LIN {X 0,Y 432.389,Z 395.501,A -85,B 0,C 180,E1 -9380.764,E2 -9380.764} C_VEL
LIN {X 0,Y 432.358,Z 395.258,A -85,B 0,C 180,E1 -9380.859,E2 -9380.859} C_VEL
LIN {X 0,Y 432.387,Z 395.255,A -85,B 0,C 180,E1 -9384.463,E2 -9384.463} C_VEL
LIN {X 0,Y 432.394,Z 395.251,A -85,B 0,C 180,E1 -9387.071,E2 -9387.071} C_VEL
LIN {X 0,Y 432.35,Z 395.255,A -85,B 0,C 180,E1 -9390.51,E2 -9390.51} C_VEL
LIN {X 0,Y 432.362,Z 395.254,A -85,B 0,C 180,E1 -9394.003,E2 -9394.003} C_VEL
LIN {X 0,Y 432.325,Z 395.26,A -85,B 0,C 180,E1 -9397.197,E2 -9397.197} C_VEL
LIN {X 0,Y 432.339,Z 395.258,A -85,B 0,C 180,E1 -9400.179,E2 -9400.179} C_VEL
LIN {X 0,Y 432.32,Z 395.262,A -85,B 0,C 180,E1 -9403.06,E2 -9403.06} C_VEL
LIN {X 0,Y 432.405,Z 395.425,A -85,B 0,C 180,E1 -9405.158,E2 -9405.158} C_VEL
LIN {X 0,Y 433.777,Z 402.089,A -85,B 0,C 180,E1 -9408.184,E2 -9408.184} C_VEL
LIN {X 0,Y 434.807,Z 407.668,A -85,B 0,C 180,E1 -9410.323,E2 -9410.323} C_VEL
LIN {X 0,Y 434.807,Z 411.22,A -85,B 0,C 180,E1 -9411.515,E2 -9411.515} C_VEL
LIN {X 0,Y 433.579,Z 424.383,A -85,B 0,C 180,E1 -9415.435,E2 -9415.435} C_VEL
LIN {X 0,Y 433.139,Z 436.415,A -85,B 0,C 180,E1 -9418.719,E2 -9418.719} C_VEL
LIN {X 0,Y 432.871,Z 446.188,A -85,B 0,C 180,E1 -9421.251,E2 -9421.251} C_VEL
LIN {X 0,Y 432.552,Z 460.292,A -85,B 0,C 180,E1 -9424.753,E2 -9424.753} C_VEL
LIN {X 0,Y 432.258,Z 473.917,A -85,B 0,C 180,E1 -9428.04,E2 -9428.04} C_VEL
LIN {X 0,Y 432.199,Z 479.961,A -85,B 0,C 180,E1 -9429.474,E2 -9429.474} C_VEL
LIN {X 0,Y 434.596,Z 497.607,A -85,B 0,C 180,E1 -9430.147,E2 -9430.147} C_VEL
LIN {X 0,Y 435.507,Z 512.403,A -85,B 0,C 180,E1 -9430.82,E2 -9430.82} C_VEL
LIN {X 0,Y 436.409,Z 524.648,A -85,B 0,C 180,E1 -9431.515,E2 -9431.515} C_VEL
LIN {X 0,Y 435.473,Z 538.641,A -85,B 0,C 180,E1 -9432.41,E2 -9432.41} C_VEL
LIN {X 0,Y 434.546,Z 551.621,A -85,B 0,C 180,E1 -9433.437,E2 -9433.437} C_VEL
LIN {X 0,Y 433.58,Z 564.986,A -85,B 0,C 180,E1 -9434.727,E2 -9434.727} C_VEL
LIN {X 0,Y 432.899,Z 577.024,A -85,B 0,C 180,E1 -9436.144,E2 -9436.144} C_VEL
LIN {X 0,Y 432.318,Z 587.05,A -85,B 0,C 180,E1 -9437.569,E2 -9437.569} C_VEL
LIN {X 0,Y 432.076,Z 595.4,A -85,B 0,C 180,E1 -9438.981,E2 -9438.981} C_VEL
LIN {X 0,Y 431.843,Z 603.466,A -85,B 0,C 180,E1 -9440.633,E2 -9440.633} C_VEL
LIN {X 0,Y 431.739,Z 609.158,A -85,B 0,C 180,E1 -9442.046,E2 -9442.046} C_VEL
LIN {X 0,Y 431.725,Z 613.768,A -85,B 0,C 180,E1 -9443.456,E2 -9443.456} C_VEL
LIN {X 0,Y 431.834,Z 618.501,A -85,B 0,C 180,E1 -9445.332,E2 -9445.332} C_VEL
LIN {X 0,Y 431.768,Z 621.63,A -85,B 0,C 180,E1 -9447.2,E2 -9447.2} C_VEL
LIN {X 0,Y 431.795,Z 623.265,A -85,B 0,C 180,E1 -9449.066,E2 -9449.066} C_VEL
LIN {X 0,Y 431.897,Z 623.543,A -85,B 0,C 180,E1 -9449.999,E2 -9449.999} C_VEL
LIN {X 0,Y 431.718,Z 622.951,A -85,B 0,C 180,E1 -9451.865,E2 -9451.865} C_VEL
LIN {X 0,Y 431.718,Z 620.927,A -85,B 0,C 180,E1 -9453.732,E2 -9453.732} C_VEL
LIN {X 0,Y 431.638,Z 617.389,A -85,B 0,C 180,E1 -9455.605,E2 -9455.605} C_VEL
LIN {X 0,Y 431.629,Z 613.716,A -85,B 0,C 180,E1 -9457.013,E2 -9457.013} C_VEL
LIN {X 0,Y 431.673,Z 609.053,A -85,B 0,C 180,E1 -9458.425,E2 -9458.425} C_VEL
LIN {X 0,Y 431.835,Z 602.28,A -85,B 0,C 180,E1 -9460.075,E2 -9460.075} C_VEL
LIN {X 0,Y 432.208,Z 593.835,A -85,B 0,C 180,E1 -9461.726,E2 -9461.726} C_VEL
LIN {X 0,Y 432.652,Z 585.027,A -85,B 0,C 180,E1 -9463.144,E2 -9463.144} C_VEL
LIN {X 0,Y 433.303,Z 574.399,A -85,B 0,C 180,E1 -9464.559,E2 -9464.559} C_VEL
LIN {X 0,Y 434.087,Z 562.586,A -85,B 0,C 180,E1 -9465.854,E2 -9465.854} C_VEL
LIN {X 0,Y 434.998,Z 550.878,A -85,B 0,C 180,E1 -9466.906,E2 -9466.906} C_VEL
LIN {X 0,Y 435.864,Z 538.135,A -85,B 0,C 180,E1 -9467.839,E2 -9467.839} C_VEL
LIN {X 0,Y 436.673,Z 523.959,A -85,B 0,C 180,E1 -9468.654,E2 -9468.654} C_VEL
LIN {X 0,Y 435.13,Z 509.071,A -85,B 0,C 180,E1 -9469.367,E2 -9469.367} C_VEL
LIN {X 0,Y 433.039,Z 493.7,A -85,B 0,C 180,E1 -9469.915,E2 -9469.915} C_VEL
LIN {X 0,Y 432.378,Z 488.684,A -85,B 0,C 180,E1 -9470.081,E2 -9470.081} C_VEL
LIN {X 0,Y 432.86,Z 475.595,A -85,B 0,C 180,E1 -9473.438,E2 -9473.438} C_VEL
LIN {X 0,Y 433.463,Z 461.986,A -85,B 0,C 180,E1 -9476.998,E2 -9476.998} C_VEL
LIN {X 0,Y 434.313,Z 447.187,A -85,B 0,C 180,E1 -9480.947,E2 -9480.947} C_VEL
LIN {X 0,Y 435.145,Z 434.082,A -85,B 0,C 180,E1 -9484.543,E2 -9484.543} C_VEL
LIN {X 0,Y 436.259,Z 419.683,A -85,B 0,C 180,E1 -9488.625,E2 -9488.625} C_VEL
LIN {X 0,Y 436.418,Z 416.038,A -85,B 0,C 180,E1 -9489.689,E2 -9489.689} C_VEL
LIN {X 0,Y 435.184,Z 408.622,A -85,B 0,C 180,E1 -9492.023,E2 -9492.023} C_VEL
LIN {X 0,Y 432.796,Z 397.532,A -85,B 0,C 180,E1 -9495.713,E2 -9495.713} C_VEL
LIN {X 0,Y 432.346,Z 395.255,A -85,B 0,C 180,E1 -9496.543,E2 -9496.543} C_VEL
LIN {X 0,Y 432.352,Z 395.257,A -85,B 0,C 180,E1 -9499.815,E2 -9499.815} C_VEL
LIN {X 0,Y 432.309,Z 395.26,A -85,B 0,C 180,E1 -9503.022,E2 -9503.022} C_VEL
LIN {X 0,Y 432.35,Z 395.253,A -85,B 0,C 180,E1 -9505.996,E2 -9505.996} C_VEL
LIN {X 0,Y 432.385,Z 395.25,A -85,B 0,C 180,E1 -9509.743,E2 -9509.743} C_VEL
LIN {X 0,Y 432.39,Z 395.252,A -85,B 0,C 180,E1 -9513.372,E2 -9513.372} C_VEL
LIN {X 0,Y 432.361,Z 395.251,A -85,B 0,C 180,E1 -9516.023,E2 -9516.023} C_VEL
LIN {X 0,Y 432.34,Z 395.257,A -85,B 0,C 180,E1 -9519.046,E2 -9519.046} C_VEL
LIN {X 0,Y 432.367,Z 395.251,A -85,B 0,C 180,E1 -9522.011,E2 -9522.011} C_VEL
LIN {X 0,Y 432.385,Z 395.251,A -85,B 0,C 180,E1 -9524.926,E2 -9524.926} C_VEL
LIN {X 0,Y 432.47,Z 395.238,A -85,B 0,C 180,E1 -9527.804,E2 -9527.804} C_VEL
LIN {X 0,Y 432.481,Z 395.238,A -85,B 0,C 180,E1 -9531.59,E2 -9531.59} C_VEL
LIN {X 0,Y 432.588,Z 395.225,A -85,B 0,C 180,E1 -9534.406,E2 -9534.406} C_VEL
LIN {X 0,Y 432.596,Z 395.223,A -85,B 0,C 180,E1 -9538.138,E2 -9538.138} C_VEL
LIN {X 0,Y 432.724,Z 395.206,A -85,B 0,C 180,E1 -9540,E2 -9540} C_VEL
LIN {X 0,Y 432.597,Z 395.224,A -85,B 0,C 180,E1 -9542.794,E2 -9542.794} C_VEL
LIN {X 0,Y 432.564,Z 395.228,A -85,B 0,C 180,E1 -9546.531,E2 -9546.531} C_VEL
LIN {X 0,Y 432.435,Z 395.244,A -85,B 0,C 180,E1 -9549.354,E2 -9549.354} C_VEL
LIN {X 0,Y 432.435,Z 395.245,A -85,B 0,C 180,E1 -9552.813,E2 -9552.813} C_VEL
LIN {X 0,Y 432.403,Z 395.248,A -85,B 0,C 180,E1 -9556.48,E2 -9556.48} C_VEL
LIN {X 0,Y 432.33,Z 395.256,A -85,B 0,C 180,E1 -9559.961,E2 -9559.961} C_VEL
LIN {X 0,Y 432.31,Z 395.262,A -85,B 0,C 180,E1 -9562.965,E2 -9562.965} C_VEL
LIN {X 0,Y 432.356,Z 395.253,A -85,B 0,C 180,E1 -9566.033,E2 -9566.033} C_VEL
LIN {X 0,Y 432.335,Z 395.256,A -85,B 0,C 180,E1 -9569.188,E2 -9569.188} C_VEL
LIN {X 0,Y 432.316,Z 395.259,A -85,B 0,C 180,E1 -9572.444,E2 -9572.444} C_VEL
LIN {X 0,Y 432.339,Z 395.254,A -85,B 0,C 180,E1 -9575.633,E2 -9575.633} C_VEL
LIN {X 0,Y 432.346,Z 395.257,A -85,B 0,C 180,E1 -9578.718,E2 -9578.718} C_VEL
LIN {X 0,Y 432.33,Z 395.256,A -85,B 0,C 180,E1 -9581.798,E2 -9581.798} C_VEL
LIN {X 0,Y 432.337,Z 395.256,A -85,B 0,C 180,E1 -9584.347,E2 -9584.347} C_VEL
LIN {X 0,Y 432.316,Z 395.259,A -85,B 0,C 180,E1 -9587.017,E2 -9587.017} C_VEL
LIN {X 0,Y 432.353,Z 395.253,A -85,B 0,C 180,E1 -9589.818,E2 -9589.818} C_VEL
LIN {X 0,Y 432.315,Z 395.259,A -85,B 0,C 180,E1 -9593.025,E2 -9593.025} C_VEL
LIN {X 0,Y 432.357,Z 395.253,A -85,B 0,C 180,E1 -9595.998,E2 -9595.998} C_VEL
LIN {X 0,Y 432.346,Z 395.253,A -85,B 0,C 180,E1 -9599.491,E2 -9599.491} C_VEL
LIN {X 0,Y 432.392,Z 395.249,A -85,B 0,C 180,E1 -9602.93,E2 -9602.93} C_VEL
LIN {X 0,Y 432.372,Z 395.252,A -85,B 0,C 180,E1 -9606.025,E2 -9606.025} C_VEL
LIN {X 0,Y 432.351,Z 395.253,A -85,B 0,C 180,E1 -9609.047,E2 -9609.047} C_VEL
LIN {X 0,Y 432.377,Z 395.251,A -85,B 0,C 180,E1 -9612.012,E2 -9612.012} C_VEL
LIN {X 0,Y 432.314,Z 395.26,A -85,B 0,C 180,E1 -9614.925,E2 -9614.925} C_VEL
LIN {X 0,Y 432.25,Z 395.365,A -85,B 0,C 180,E1 -9616.547,E2 -9616.547} C_VEL
LIN {X 0,Y 436.298,Z 408.442,A -85,B 0,C 180,E1 -9617.107,E2 -9617.107} C_VEL
LIN {X 0,Y 436.567,Z 411.618,A -85,B 0,C 180,E1 -9617.251,E2 -9617.251} C_VEL
LIN {X 0,Y 436.282,Z 423.378,A -85,B 0,C 180,E1 -9617.832,E2 -9617.832} C_VEL
LIN {X 0,Y 435.847,Z 435.168,A -85,B 0,C 180,E1 -9618.609,E2 -9618.609} C_VEL
LIN {X 0,Y 435.323,Z 446.119,A -85,B 0,C 180,E1 -9619.537,E2 -9619.537} C_VEL
LIN {X 0,Y 434.762,Z 455.934,A -85,B 0,C 180,E1 -9620.569,E2 -9620.569} C_VEL
LIN {X 0,Y 434.12,Z 465.767,A -85,B 0,C 180,E1 -9621.858,E2 -9621.858} C_VEL
LIN {X 0,Y 433.656,Z 474.255,A -85,B 0,C 180,E1 -9623.253,E2 -9623.253} C_VEL
LIN {X 0,Y 433.113,Z 481.113,A -85,B 0,C 180,E1 -9624.647,E2 -9624.647} C_VEL
LIN {X 0,Y 432.913,Z 485.709,A -85,B 0,C 180,E1 -9625.812,E2 -9625.812} C_VEL
LIN {X 0,Y 432.731,Z 487.452,A -85,B 0,C 180,E1 -9626.316,E2 -9626.316} C_VEL
LIN {X 0,Y 431.918,Z 489.8,A -85,B 0,C 180,E1 -9627.029,E2 -9627.029} C_VEL
LIN {X 0,Y 427.594,Z 494.515,A -85,B 0,C 180,E1 -9628.67,E2 -9628.67} C_VEL
LIN {X 0,Y 425.543,Z 496.535,A -85,B 0,C 180,E1 -9629.661,E2 -9629.661} C_VEL
LIN {X 0,Y 425.142,Z 497.269,A -85,B 0,C 180,E1 -9630.181,E2 -9630.181} C_VEL
LIN {X 0,Y 425.026,Z 498.178,A -85,B 0,C 180,E1 -9630.948,E2 -9630.948} C_VEL
LIN {X 0,Y 425.094,Z 498.851,A -85,B 0,C 180,E1 -9631.896,E2 -9631.896} C_VEL
LIN {X 0,Y 425.025,Z 499.13,A -85,B 0,C 180,E1 -9633.793,E2 -9633.793} C_VEL
LIN {X 0,Y 425.111,Z 498.668,A -85,B 0,C 180,E1 -9634.742,E2 -9634.742} C_VEL
LIN {X 0,Y 425.3,Z 497.792,A -85,B 0,C 180,E1 -9635.691,E2 -9635.691} C_VEL
LIN {X 0,Y 425.456,Z 494.927,A -85,B 0,C 180,E1 -9637.595,E2 -9637.595} C_VEL
LIN {X 0,Y 425.736,Z 491.621,A -85,B 0,C 180,E1 -9639.024,E2 -9639.024} C_VEL
LIN {X 0,Y 426.167,Z 487.23,A -85,B 0,C 180,E1 -9640.452,E2 -9640.452} C_VEL
LIN {X 0,Y 426.614,Z 480.562,A -85,B 0,C 180,E1 -9642.126,E2 -9642.126} C_VEL
LIN {X 0,Y 426.971,Z 474.618,A -85,B 0,C 180,E1 -9643.324,E2 -9643.324} C_VEL
LIN {X 0,Y 427.736,Z 465.841,A -85,B 0,C 180,E1 -9644.755,E2 -9644.755} C_VEL
LIN {X 0,Y 428.389,Z 455.68,A -85,B 0,C 180,E1 -9646.073,E2 -9646.073} C_VEL
LIN {X 0,Y 428.99,Z 445.34,A -85,B 0,C 180,E1 -9647.152,E2 -9647.152} C_VEL
LIN {X 0,Y 429.538,Z 435.288,A -85,B 0,C 180,E1 -9647.989,E2 -9647.989} C_VEL
LIN {X 0,Y 430.03,Z 423.551,A -85,B 0,C 180,E1 -9648.754,E2 -9648.754} C_VEL
LIN {X 0,Y 430.232,Z 411.232,A -85,B 0,C 180,E1 -9649.362,E2 -9649.362} C_VEL
LIN {X 0,Y 426.035,Z 398.909,A -85,B 0,C 180,E1 -9649.98,E2 -9649.98} C_VEL
LIN {X 0,Y 425.159,Z 396.153,A -85,B 0,C 180,E1 -9650.101,E2 -9650.101} C_VEL
LIN {X 0,Y 425.287,Z 396.134,A -85,B 0,C 180,E1 -9653.367,E2 -9653.367} C_VEL
LIN {X 0,Y 425.361,Z 396.125,A -85,B 0,C 180,E1 -9656.495,E2 -9656.495} C_VEL
LIN {X 0,Y 425.297,Z 396.133,A -85,B 0,C 180,E1 -9659.72,E2 -9659.72} C_VEL
LIN {X 0,Y 425.287,Z 396.139,A -85,B 0,C 180,E1 -9663.048,E2 -9663.048} C_VEL
LIN {X 0,Y 425.287,Z 396.135,A -85,B 0,C 180,E1 -9665.929,E2 -9665.929} C_VEL
LIN {X 0,Y 425.293,Z 396.129,A -85,B 0,C 180,E1 -9669.042,E2 -9669.042} C_VEL
LIN {X 0,Y 425.295,Z 396.132,A -85,B 0,C 180,E1 -9671.958,E2 -9671.958} C_VEL
LIN {X 0,Y 425.295,Z 396.128,A -85,B 0,C 180,E1 -9675.283,E2 -9675.283} C_VEL
LIN {X 0,Y 425.281,Z 396.131,A -85,B 0,C 180,E1 -9678.622,E2 -9678.622} C_VEL
LIN {X 0,Y 425.314,Z 396.108,A -85,B 0,C 180,E1 -9681.103,E2 -9681.103} C_VEL
LIN {X 0,Y 425.306,Z 396.131,A -85,B 0,C 180,E1 -9684.664,E2 -9684.664} C_VEL
LIN {X 0,Y 425.269,Z 396.125,A -85,B 0,C 180,E1 -9688.073,E2 -9688.073} C_VEL
LIN {X 0,Y 425.335,Z 396.103,A -85,B 0,C 180,E1 -9691.368,E2 -9691.368} C_VEL
LIN {X 0,Y 425.358,Z 396.118,A -85,B 0,C 180,E1 -9693.505,E2 -9693.505} C_VEL
LIN {X 0,Y 425.289,Z 396.132,A -85,B 0,C 180,E1 -9696.633,E2 -9696.633} C_VEL
LIN {X 0,Y 425.299,Z 396.135,A -85,B 0,C 180,E1 -9699.694,E2 -9699.694} C_VEL
LIN {X 0,Y 425.329,Z 396.131,A -85,B 0,C 180,E1 -9701.889,E2 -9701.889} C_VEL
LIN {X 0,Y 430.063,Z 411.616,A -85,B 0,C 180,E1 -9703.015,E2 -9703.015} C_VEL
LIN {X 0,Y 430.272,Z 415.083,A -85,B 0,C 180,E1 -9703.268,E2 -9703.268} C_VEL
LIN {X 0,Y 429.619,Z 427.403,A -85,B 0,C 180,E1 -9704.219,E2 -9704.219} C_VEL
LIN {X 0,Y 428.793,Z 440.383,A -85,B 0,C 180,E1 -9705.449,E2 -9705.449} C_VEL
LIN {X 0,Y 428.002,Z 451.242,A -85,B 0,C 180,E1 -9706.709,E2 -9706.709} C_VEL
LIN {X 0,Y 427.252,Z 461.376,A -85,B 0,C 180,E1 -9708.134,E2 -9708.134} C_VEL
LIN {X 0,Y 426.771,Z 469.803,A -85,B 0,C 180,E1 -9709.563,E2 -9709.563} C_VEL
LIN {X 0,Y 426.188,Z 477.894,A -85,B 0,C 180,E1 -9711.226,E2 -9711.226} C_VEL
LIN {X 0,Y 425.775,Z 484.425,A -85,B 0,C 180,E1 -9712.888,E2 -9712.888} C_VEL
LIN {X 0,Y 425.45,Z 490.251,A -85,B 0,C 180,E1 -9714.787,E2 -9714.787} C_VEL
LIN {X 0,Y 425.156,Z 493.572,A -85,B 0,C 180,E1 -9716.208,E2 -9716.208} C_VEL
LIN {X 0,Y 425.096,Z 496.722,A -85,B 0,C 180,E1 -9718.105,E2 -9718.105} C_VEL
LIN {X 0,Y 425.055,Z 498.526,A -85,B 0,C 180,E1 -9720,E2 -9720} C_VEL
LIN {X 0,Y 425.159,Z 498.985,A -85,B 0,C 180,E1 -9721.894,E2 -9721.894} C_VEL
LIN {X 0,Y 425.197,Z 498.132,A -85,B 0,C 180,E1 -9723.791,E2 -9723.791} C_VEL
LIN {X 0,Y 425.467,Z 495.878,A -85,B 0,C 180,E1 -9725.688,E2 -9725.688} C_VEL
LIN {X 0,Y 425.857,Z 492.193,A -85,B 0,C 180,E1 -9727.586,E2 -9727.586} C_VEL
LIN {X 0,Y 426.379,Z 487.005,A -85,B 0,C 180,E1 -9729.487,E2 -9729.487} C_VEL
LIN {X 0,Y 426.836,Z 481.998,A -85,B 0,C 180,E1 -9730.915,E2 -9730.915} C_VEL
LIN {X 0,Y 427.533,Z 474.75,A -85,B 0,C 180,E1 -9732.58,E2 -9732.58} C_VEL
LIN {X 0,Y 428.349,Z 467.101,A -85,B 0,C 180,E1 -9734.005,E2 -9734.005} C_VEL
LIN {X 0,Y 429.177,Z 457.883,A -85,B 0,C 180,E1 -9735.432,E2 -9735.432} C_VEL
LIN {X 0,Y 430.005,Z 447.738,A -85,B 0,C 180,E1 -9736.742,E2 -9736.742} C_VEL
LIN {X 0,Y 430.927,Z 436.514,A -85,B 0,C 180,E1 -9737.929,E2 -9737.929} C_VEL
LIN {X 0,Y 431.776,Z 424.026,A -85,B 0,C 180,E1 -9738.998,E2 -9738.998} C_VEL
LIN {X 0,Y 432.22,Z 415.031,A -85,B 0,C 180,E1 -9739.645,E2 -9739.645} C_VEL
LIN {X 0,Y 428.671,Z 404.666,A -85,B 0,C 180,E1 -9740.551,E2 -9740.551} C_VEL
LIN {X 0,Y 425.717,Z 397.734,A -85,B 0,C 180,E1 -9741.139,E2 -9741.139} C_VEL
LIN {X 0,Y 425.315,Z 396.136,A -85,B 0,C 180,E1 -9741.263,E2 -9741.263} C_VEL
LIN {X 0,Y 425.329,Z 396.134,A -85,B 0,C 180,E1 -9744.659,E2 -9744.659} C_VEL
LIN {X 0,Y 425.352,Z 396.129,A -85,B 0,C 180,E1 -9747.557,E2 -9747.557} C_VEL
LIN {X 0,Y 425.291,Z 396.136,A -85,B 0,C 180,E1 -9750.816,E2 -9750.816} C_VEL
LIN {X 0,Y 425.314,Z 396.134,A -85,B 0,C 180,E1 -9754.288,E2 -9754.288} C_VEL
LIN {X 0,Y 425.282,Z 396.137,A -85,B 0,C 180,E1 -9757.694,E2 -9757.694} C_VEL
LIN {X 0,Y 425.284,Z 396.137,A -85,B 0,C 180,E1 -9760.52,E2 -9760.52} C_VEL
LIN {X 0,Y 425.261,Z 396.14,A -85,B 0,C 180,E1 -9763.35,E2 -9763.35} C_VEL
LIN {X 0,Y 425.325,Z 396.216,A -85,B 0,C 180,E1 -9764.493,E2 -9764.493} C_VEL
LIN {X 0,Y 426.623,Z 402.454,A -85,B 0,C 180,E1 -9767.513,E2 -9767.513} C_VEL
LIN {X 0,Y 427.871,Z 409.046,A -85,B 0,C 180,E1 -9770.163,E2 -9770.163} C_VEL
LIN {X 0,Y 427.932,Z 412.57,A -85,B 0,C 180,E1 -9771.384,E2 -9771.384} C_VEL
LIN {X 0,Y 426.652,Z 424.987,A -85,B 0,C 180,E1 -9775.182,E2 -9775.182} C_VEL
LIN {X 0,Y 426.184,Z 435.513,A -85,B 0,C 180,E1 -9778.149,E2 -9778.149} C_VEL
LIN {X 0,Y 425.843,Z 446.252,A -85,B 0,C 180,E1 -9781.009,E2 -9781.009} C_VEL
LIN {X 0,Y 425.484,Z 460.214,A -85,B 0,C 180,E1 -9784.566,E2 -9784.566} C_VEL
LIN {X 0,Y 425.213,Z 473.159,A -85,B 0,C 180,E1 -9787.756,E2 -9787.756} C_VEL
LIN {X 0,Y 425.138,Z 478.361,A -85,B 0,C 180,E1 -9789.022,E2 -9789.022} C_VEL
LIN {X 0,Y 427.643,Z 495.642,A -85,B 0,C 180,E1 -9789.714,E2 -9789.714} C_VEL
LIN {X 0,Y 428.624,Z 510.852,A -85,B 0,C 180,E1 -9790.432,E2 -9790.432} C_VEL
LIN {X 0,Y 429.347,Z 521.991,A -85,B 0,C 180,E1 -9791.075,E2 -9791.075} C_VEL
LIN {X 0,Y 429.428,Z 526.944,A -85,B 0,C 180,E1 -9791.388,E2 -9791.388} C_VEL
LIN {X 0,Y 428.355,Z 541.511,A -85,B 0,C 180,E1 -9792.395,E2 -9792.395} C_VEL
LIN {X 0,Y 427.386,Z 554.595,A -85,B 0,C 180,E1 -9793.52,E2 -9793.52} C_VEL
LIN {X 0,Y 426.442,Z 567.153,A -85,B 0,C 180,E1 -9794.832,E2 -9794.832} C_VEL
LIN {X 0,Y 425.786,Z 577.68,A -85,B 0,C 180,E1 -9796.152,E2 -9796.152} C_VEL
LIN {X 0,Y 425.232,Z 587.356,A -85,B 0,C 180,E1 -9797.592,E2 -9797.592} C_VEL
LIN {X 0,Y 424.924,Z 596.74,A -85,B 0,C 180,E1 -9799.276,E2 -9799.276} C_VEL
LIN {X 0,Y 424.744,Z 604.38,A -85,B 0,C 180,E1 -9800.955,E2 -9800.955} C_VEL
LIN {X 0,Y 424.645,Z 609.69,A -85,B 0,C 180,E1 -9802.391,E2 -9802.391} C_VEL
LIN {X 0,Y 424.668,Z 614.036,A -85,B 0,C 180,E1 -9803.824,E2 -9803.824} C_VEL
LIN {X 0,Y 424.783,Z 617.441,A -85,B 0,C 180,E1 -9805.254,E2 -9805.254} C_VEL
LIN {X 0,Y 424.732,Z 620.584,A -85,B 0,C 180,E1 -9807.154,E2 -9807.154} C_VEL
LIN {X 0,Y 424.789,Z 622.227,A -85,B 0,C 180,E1 -9809.051,E2 -9809.051} C_VEL
LIN {X 0,Y 424.878,Z 622.505,A -85,B 0,C 180,E1 -9809.999,E2 -9809.999} C_VEL
LIN {X 0,Y 424.687,Z 621.912,A -85,B 0,C 180,E1 -9811.896,E2 -9811.896} C_VEL
LIN {X 0,Y 424.68,Z 619.88,A -85,B 0,C 180,E1 -9813.794,E2 -9813.794} C_VEL
LIN {X 0,Y 424.589,Z 616.327,A -85,B 0,C 180,E1 -9815.699,E2 -9815.699} C_VEL
LIN {X 0,Y 424.563,Z 612.627,A -85,B 0,C 180,E1 -9817.13,E2 -9817.13} C_VEL
LIN {X 0,Y 424.614,Z 607.956,A -85,B 0,C 180,E1 -9818.566,E2 -9818.566} C_VEL
LIN {X 0,Y 424.778,Z 601.144,A -85,B 0,C 180,E1 -9820.244,E2 -9820.244} C_VEL
LIN {X 0,Y 425.186,Z 592.649,A -85,B 0,C 180,E1 -9821.923,E2 -9821.923} C_VEL
LIN {X 0,Y 425.629,Z 583.787,A -85,B 0,C 180,E1 -9823.365,E2 -9823.365} C_VEL
LIN {X 0,Y 426.359,Z 573.112,A -85,B 0,C 180,E1 -9824.802,E2 -9824.802} C_VEL
LIN {X 0,Y 427.079,Z 562.4,A -85,B 0,C 180,E1 -9825.999,E2 -9825.999} C_VEL
LIN {X 0,Y 428.013,Z 550.85,A -85,B 0,C 180,E1 -9827.067,E2 -9827.067} C_VEL
LIN {X 0,Y 428.896,Z 538.283,A -85,B 0,C 180,E1 -9828.018,E2 -9828.018} C_VEL
LIN {X 0,Y 429.747,Z 524.556,A -85,B 0,C 180,E1 -9828.842,E2 -9828.842} C_VEL
LIN {X 0,Y 428.29,Z 510.13,A -85,B 0,C 180,E1 -9829.571,E2 -9829.571} C_VEL
LIN {X 0,Y 426.298,Z 495.12,A -85,B 0,C 180,E1 -9830.144,E2 -9830.144} C_VEL
LIN {X 0,Y 425.299,Z 487.926,A -85,B 0,C 180,E1 -9830.367,E2 -9830.367} C_VEL
LIN {X 0,Y 425.837,Z 474.659,A -85,B 0,C 180,E1 -9833.849,E2 -9833.849} C_VEL
LIN {X 0,Y 426.506,Z 461.05,A -85,B 0,C 180,E1 -9837.475,E2 -9837.475} C_VEL
LIN {X 0,Y 427.325,Z 447.321,A -85,B 0,C 180,E1 -9841.216,E2 -9841.216} C_VEL
LIN {X 0,Y 428.091,Z 435.963,A -85,B 0,C 180,E1 -9844.389,E2 -9844.389} C_VEL
LIN {X 0,Y 429.256,Z 421.756,A -85,B 0,C 180,E1 -9848.472,E2 -9848.472} C_VEL
LIN {X 0,Y 429.497,Z 417.526,A -85,B 0,C 180,E1 -9849.729,E2 -9849.729} C_VEL
LIN {X 0,Y 428.127,Z 409.471,A -85,B 0,C 180,E1 -9852.3,E2 -9852.3} C_VEL
LIN {X 0,Y 426.022,Z 399.626,A -85,B 0,C 180,E1 -9855.628,E2 -9855.628} C_VEL
LIN {X 0,Y 425.333,Z 396.129,A -85,B 0,C 180,E1 -9856.917,E2 -9856.917} C_VEL
LIN {X 0,Y 425.305,Z 396.135,A -85,B 0,C 180,E1 -9859.875,E2 -9859.875} C_VEL
LIN {X 0,Y 425.279,Z 396.135,A -85,B 0,C 180,E1 -9862.486,E2 -9862.486} C_VEL
LIN {X 0,Y 425.299,Z 396.132,A -85,B 0,C 180,E1 -9865.817,E2 -9865.817} C_VEL
LIN {X 0,Y 425.291,Z 396.136,A -85,B 0,C 180,E1 -9869.236,E2 -9869.236} C_VEL
LIN {X 0,Y 425.34,Z 396.126,A -85,B 0,C 180,E1 -9872.442,E2 -9872.442} C_VEL
LIN {X 0,Y 425.341,Z 396.128,A -85,B 0,C 180,E1 -9875.602,E2 -9875.602} C_VEL
LIN {X 0,Y 425.283,Z 396.135,A -85,B 0,C 180,E1 -9878.681,E2 -9878.681} C_VEL
LIN {X 0,Y 425.322,Z 396.129,A -85,B 0,C 180,E1 -9881.702,E2 -9881.702} C_VEL
LIN {X 0,Y 425.338,Z 396.128,A -85,B 0,C 180,E1 -9884.67,E2 -9884.67} C_VEL
LIN {X 0,Y 425.419,Z 396.117,A -85,B 0,C 180,E1 -9887.599,E2 -9887.599} C_VEL
LIN {X 0,Y 425.432,Z 396.116,A -85,B 0,C 180,E1 -9891.45,E2 -9891.45} C_VEL
LIN {X 0,Y 425.544,Z 396.101,A -85,B 0,C 180,E1 -9894.313,E2 -9894.313} C_VEL
LIN {X 0,Y 425.565,Z 396.098,A -85,B 0,C 180,E1 -9898.107,E2 -9898.107} C_VEL
LIN {X 0,Y 425.694,Z 396.082,A -85,B 0,C 180,E1 -9900,E2 -9900} C_VEL
LIN {X 0,Y 425.548,Z 396.103,A -85,B 0,C 180,E1 -9902.84,E2 -9902.84} C_VEL
LIN {X 0,Y 425.521,Z 396.105,A -85,B 0,C 180,E1 -9906.648,E2 -9906.648} C_VEL
LIN {X 0,Y 425.394,Z 396.12,A -85,B 0,C 180,E1 -9909.51,E2 -9909.51} C_VEL
LIN {X 0,Y 425.394,Z 396.123,A -85,B 0,C 180,E1 -9912.911,E2 -9912.911} C_VEL
LIN {X 0,Y 425.351,Z 396.127,A -85,B 0,C 180,E1 -9916.606,E2 -9916.606} C_VEL
LIN {X 0,Y 425.319,Z 396.128,A -85,B 0,C 180,E1 -9919.637,E2 -9919.637} C_VEL
LIN {X 0,Y 425.298,Z 396.132,A -85,B 0,C 180,E1 -9923.366,E2 -9923.366} C_VEL
LIN {X 0,Y 425.34,Z 396.13,A -85,B 0,C 180,E1 -9926.846,E2 -9926.846} C_VEL
LIN {X 0,Y 425.283,Z 396.133,A -85,B 0,C 180,E1 -9929.721,E2 -9929.721} C_VEL
LIN {X 0,Y 425.275,Z 396.137,A -85,B 0,C 180,E1 -9933.049,E2 -9933.049} C_VEL
LIN {X 0,Y 425.278,Z 396.134,A -85,B 0,C 180,E1 -9935.93,E2 -9935.93} C_VEL
LIN {X 0,Y 425.297,Z 396.133,A -85,B 0,C 180,E1 -9939.046,E2 -9939.046} C_VEL
LIN {X 0,Y 425.273,Z 396.138,A -85,B 0,C 180,E1 -9942.654,E2 -9942.654} C_VEL
LIN {X 0,Y 425.257,Z 396.138,A -85,B 0,C 180,E1 -9946.046,E2 -9946.046} C_VEL
LIN {X 0,Y 425.301,Z 396.135,A -85,B 0,C 180,E1 -9948.626,E2 -9948.626} C_VEL
LIN {X 0,Y 425.321,Z 396.129,A -85,B 0,C 180,E1 -9951.106,E2 -9951.106} C_VEL
LIN {X 0,Y 425.298,Z 396.136,A -85,B 0,C 180,E1 -9954.666,E2 -9954.666} C_VEL
LIN {X 0,Y 425.264,Z 396.137,A -85,B 0,C 180,E1 -9958.075,E2 -9958.075} C_VEL
LIN {X 0,Y 425.33,Z 396.127,A -85,B 0,C 180,E1 -9961.369,E2 -9961.369} C_VEL
LIN {X 0,Y 425.296,Z 396.136,A -85,B 0,C 180,E1 -9964.556,E2 -9964.556} C_VEL
LIN {X 0,Y 425.288,Z 396.133,A -85,B 0,C 180,E1 -9967.663,E2 -9967.663} C_VEL
LIN {X 0,Y 425.363,Z 396.126,A -85,B 0,C 180,E1 -9970.705,E2 -9970.705} C_VEL
LIN {X 0,Y 425.334,Z 396.128,A -85,B 0,C 180,E1 -9973.687,E2 -9973.687} C_VEL
LIN {X 0,Y 425.256,Z 396.3,A -85,B 0,C 180,E1 -9976.286,E2 -9976.286} C_VEL
LIN {X 0,Y 429.293,Z 409.175,A -85,B 0,C 180,E1 -9976.849,E2 -9976.849} C_VEL
LIN {X 0,Y 429.763,Z 412.44,A -85,B 0,C 180,E1 -9977.006,E2 -9977.006} C_VEL
LIN {X 0,Y 429.437,Z 424.988,A -85,B 0,C 180,E1 -9977.637,E2 -9977.637} C_VEL
LIN {X 0,Y 428.99,Z 436.577,A -85,B 0,C 180,E1 -9978.424,E2 -9978.424} C_VEL
LIN {X 0,Y 428.466,Z 447.452,A -85,B 0,C 180,E1 -9979.367,E2 -9979.367} C_VEL
LIN {X 0,Y 427.856,Z 457.216,A -85,B 0,C 180,E1 -9980.416,E2 -9980.416} C_VEL
LIN {X 0,Y 427.196,Z 466.983,A -85,B 0,C 180,E1 -9981.725,E2 -9981.725} C_VEL
LIN {X 0,Y 426.707,Z 475.436,A -85,B 0,C 180,E1 -9983.143,E2 -9983.143} C_VEL
LIN {X 0,Y 426.135,Z 482.256,A -85,B 0,C 180,E1 -9984.559,E2 -9984.559} C_VEL
LIN {X 0,Y 425.924,Z 486.833,A -85,B 0,C 180,E1 -9985.743,E2 -9985.743} C_VEL
LIN {X 0,Y 425.589,Z 491.28,A -85,B 0,C 180,E1 -9987.161,E2 -9987.161} C_VEL
LIN {X 0,Y 425.415,Z 493.634,A -85,B 0,C 180,E1 -9988.108,E2 -9988.108} C_VEL
LIN {X 0,Y 425.181,Z 497.057,A -85,B 0,C 180,E1 -9990.001,E2 -9990.001} C_VEL
LIN {X 0,Y 425.142,Z 497.269,A -85,B 0,C 180,E1 -9990.181,E2 -9990.181} C_VEL
LIN {X 0,Y 424.362,Z 498.285,A -85,B 0,C 180,E1 -9990.961,E2 -9990.961} C_VEL
LIN {X 0,Y 421.437,Z 499.539,A -85,B 0,C 180,E1 -9992.235,E2 -9992.235} C_VEL
LIN {X 0,Y 419.062,Z 500.063,A -85,B 0,C 180,E1 -9993.266,E2 -9993.266} C_VEL
LIN {X 0,Y 418.09,Z 500.039,A -85,B 0,C 180,E1 -9994.065,E2 -9994.065} C_VEL
LIN {X 0,Y 418.034,Z 499.89,A -85,B 0,C 180,E1 -9994.335,E2 -9994.335} C_VEL
LIN {X 0,Y 418.3,Z 498.758,A -85,B 0,C 180,E1 -9995.787,E2 -9995.787} C_VEL
LIN {X 0,Y 418.345,Z 497.517,A -85,B 0,C 180,E1 -9996.754,E2 -9996.754} C_VEL
LIN {X 0,Y 418.564,Z 494.849,A -85,B 0,C 180,E1 -9998.206,E2 -9998.206} C_VEL
LIN {X 0,Y 418.964,Z 491.162,A -85,B 0,C 180,E1 -9999.658,E2 -9999.658} C_VEL
LIN {X 0,Y 419.375,Z 486.376,A -85,B 0,C 180,E1 -10001.113,E2 -10001.113} C_VEL
LIN {X 0,Y 419.804,Z 480.331,A -85,B 0,C 180,E1 -10002.571,E2 -10002.571} C_VEL
LIN {X 0,Y 420.299,Z 473.541,A -85,B 0,C 180,E1 -10003.889,E2 -10003.889} C_VEL
LIN {X 0,Y 420.991,Z 464.897,A -85,B 0,C 180,E1 -10005.245,E2 -10005.245} C_VEL
LIN {X 0,Y 421.658,Z 455.364,A -85,B 0,C 180,E1 -10006.461,E2 -10006.461} C_VEL
LIN {X 0,Y 422.323,Z 444.624,A -85,B 0,C 180,E1 -10007.556,E2 -10007.556} C_VEL
LIN {X 0,Y 422.844,Z 434.126,A -85,B 0,C 180,E1 -10008.41,E2 -10008.41} C_VEL
LIN {X 0,Y 423.389,Z 422.192,A -85,B 0,C 180,E1 -10009.162,E2 -10009.162} C_VEL
LIN {X 0,Y 423.366,Z 412.372,A -85,B 0,C 180,E1 -10009.647,E2 -10009.647} C_VEL
LIN {X 0,Y 419.152,Z 400.246,A -85,B 0,C 180,E1 -10010.276,E2 -10010.276} C_VEL
LIN {X 0,Y 418.131,Z 397.029,A -85,B 0,C 180,E1 -10010.421,E2 -10010.421} C_VEL
LIN {X 0,Y 418.28,Z 397.006,A -85,B 0,C 180,E1 -10013.782,E2 -10013.782} C_VEL
LIN {X 0,Y 418.316,Z 397.005,A -85,B 0,C 180,E1 -10017.071,E2 -10017.071} C_VEL
LIN {X 0,Y 418.251,Z 397.012,A -85,B 0,C 180,E1 -10020.272,E2 -10020.272} C_VEL
LIN {X 0,Y 418.253,Z 397.011,A -85,B 0,C 180,E1 -10023.678,E2 -10023.678} C_VEL
LIN {X 0,Y 418.245,Z 397.005,A -85,B 0,C 180,E1 -10027.224,E2 -10027.224} C_VEL
LIN {X 0,Y 418.252,Z 397.005,A -85,B 0,C 180,E1 -10029.683,E2 -10029.683} C_VEL
LIN {X 0,Y 418.235,Z 397.012,A -85,B 0,C 180,E1 -10032.321,E2 -10032.321} C_VEL
LIN {X 0,Y 418.245,Z 397.007,A -85,B 0,C 180,E1 -10035.109,E2 -10035.109} C_VEL
LIN {X 0,Y 418.262,Z 397.009,A -85,B 0,C 180,E1 -10037.769,E2 -10037.769} C_VEL
LIN {X 0,Y 418.262,Z 396.986,A -85,B 0,C 180,E1 -10041.559,E2 -10041.559} C_VEL
LIN {X 0,Y 418.265,Z 397.007,A -85,B 0,C 180,E1 -10045.159,E2 -10045.159} C_VEL
LIN {X 0,Y 418.25,Z 397.007,A -85,B 0,C 180,E1 -10047.472,E2 -10047.472} C_VEL
LIN {X 0,Y 418.273,Z 396.98,A -85,B 0,C 180,E1 -10050.895,E2 -10050.895} C_VEL
LIN {X 0,Y 418.273,Z 397.008,A -85,B 0,C 180,E1 -10054.096,E2 -10054.096} C_VEL
LIN {X 0,Y 418.236,Z 397.013,A -85,B 0,C 180,E1 -10057.263,E2 -10057.263} C_VEL
LIN {X 0,Y 418.287,Z 397.005,A -85,B 0,C 180,E1 -10060.364,E2 -10060.364} C_VEL
LIN {X 0,Y 418.29,Z 397.029,A -85,B 0,C 180,E1 -10061.637,E2 -10061.637} C_VEL
LIN {X 0,Y 422.19,Z 409.933,A -85,B 0,C 180,E1 -10062.564,E2 -10062.564} C_VEL
LIN {X 0,Y 423.442,Z 414.209,A -85,B 0,C 180,E1 -10062.908,E2 -10062.908} C_VEL
LIN {X 0,Y 422.789,Z 427.769,A -85,B 0,C 180,E1 -10063.957,E2 -10063.957} C_VEL
LIN {X 0,Y 422.022,Z 439.385,A -85,B 0,C 180,E1 -10065.056,E2 -10065.056} C_VEL
LIN {X 0,Y 421.344,Z 449.852,A -85,B 0,C 180,E1 -10066.249,E2 -10066.249} C_VEL
LIN {X 0,Y 420.447,Z 460.456,A -85,B 0,C 180,E1 -10067.694,E2 -10067.694} C_VEL
LIN {X 0,Y 419.912,Z 469.221,A -85,B 0,C 180,E1 -10069.147,E2 -10069.147} C_VEL
LIN {X 0,Y 419.286,Z 477.649,A -85,B 0,C 180,E1 -10070.837,E2 -10070.837} C_VEL
LIN {X 0,Y 418.911,Z 483.565,A -85,B 0,C 180,E1 -10072.287,E2 -10072.287} C_VEL
LIN {X 0,Y 418.584,Z 488.422,A -85,B 0,C 180,E1 -10073.734,E2 -10073.734} C_VEL
LIN {X 0,Y 418.348,Z 493.504,A -85,B 0,C 180,E1 -10075.664,E2 -10075.664} C_VEL
LIN {X 0,Y 418.021,Z 496.313,A -85,B 0,C 180,E1 -10077.109,E2 -10077.109} C_VEL
LIN {X 0,Y 418.077,Z 497.73,A -85,B 0,C 180,E1 -10078.073,E2 -10078.073} C_VEL
LIN {X 0,Y 418.05,Z 499.574,A -85,B 0,C 180,E1 -10080,E2 -10080} C_VEL
LIN {X 0,Y 418.165,Z 500.07,A -85,B 0,C 180,E1 -10081.926,E2 -10081.926} C_VEL
LIN {X 0,Y 418.199,Z 499.261,A -85,B 0,C 180,E1 -10083.854,E2 -10083.854} C_VEL
LIN {X 0,Y 418.499,Z 497.06,A -85,B 0,C 180,E1 -10085.783,E2 -10085.783} C_VEL
LIN {X 0,Y 418.948,Z 493.428,A -85,B 0,C 180,E1 -10087.712,E2 -10087.712} C_VEL
LIN {X 0,Y 419.502,Z 488.275,A -85,B 0,C 180,E1 -10089.644,E2 -10089.644} C_VEL
LIN {X 0,Y 419.983,Z 483.298,A -85,B 0,C 180,E1 -10091.095,E2 -10091.095} C_VEL
LIN {X 0,Y 420.729,Z 476.083,A -85,B 0,C 180,E1 -10092.787,E2 -10092.787} C_VEL
LIN {X 0,Y 421.609,Z 468.523,A -85,B 0,C 180,E1 -10094.233,E2 -10094.233} C_VEL
LIN {X 0,Y 422.506,Z 459.42,A -85,B 0,C 180,E1 -10095.682,E2 -10095.682} C_VEL
LIN {X 0,Y 423.302,Z 450.317,A -85,B 0,C 180,E1 -10096.891,E2 -10096.891} C_VEL
LIN {X 0,Y 424.229,Z 439.395,A -85,B 0,C 180,E1 -10098.097,E2 -10098.097} C_VEL
LIN {X 0,Y 425.172,Z 427.493,A -85,B 0,C 180,E1 -10099.179,E2 -10099.179} C_VEL
LIN {X 0,Y 425.841,Z 418.113,A -85,B 0,C 180,E1 -10099.879,E2 -10099.879} C_VEL
LIN {X 0,Y 423.934,Z 411.251,A -85,B 0,C 180,E1 -10100.5,E2 -10100.5} C_VEL
LIN {X 0,Y 419.888,Z 401.259,A -85,B 0,C 180,E1 -10101.401,E2 -10101.401} C_VEL
LIN {X 0,Y 418.32,Z 397.389,A -85,B 0,C 180,E1 -10101.727,E2 -10101.727} C_VEL
LIN {X 0,Y 418.237,Z 397.019,A -85,B 0,C 180,E1 -10101.79,E2 -10101.79} C_VEL
LIN {X 0,Y 418.287,Z 397.011,A -85,B 0,C 180,E1 -10104.864,E2 -10104.864} C_VEL
LIN {X 0,Y 418.294,Z 397.006,A -85,B 0,C 180,E1 -10108.063,E2 -10108.063} C_VEL
LIN {X 0,Y 418.215,Z 397.018,A -85,B 0,C 180,E1 -10111.396,E2 -10111.396} C_VEL
LIN {X 0,Y 418.268,Z 397.011,A -85,B 0,C 180,E1 -10114.58,E2 -10114.58} C_VEL
LIN {X 0,Y 418.231,Z 397.014,A -85,B 0,C 180,E1 -10117.833,E2 -10117.833} C_VEL
LIN {X 0,Y 418.225,Z 397.017,A -85,B 0,C 180,E1 -10120.948,E2 -10120.948} C_VEL
LIN {X 0,Y 418.245,Z 397.066,A -85,B 0,C 180,E1 -10123.801,E2 -10123.801} C_VEL
LIN {X 0,Y 419.385,Z 402.43,A -85,B 0,C 180,E1 -10126.6,E2 -10126.6} C_VEL
LIN {X 0,Y 420.641,Z 408.744,A -85,B 0,C 180,E1 -10129.336,E2 -10129.336} C_VEL
LIN {X 0,Y 421.104,Z 412.177,A -85,B 0,C 180,E1 -10130.639,E2 -10130.639} C_VEL
LIN {X 0,Y 420.752,Z 415.696,A -85,B 0,C 180,E1 -10131.827,E2 -10131.827} C_VEL
LIN {X 0,Y 419.632,Z 426.835,A -85,B 0,C 180,E1 -10135.289,E2 -10135.289} C_VEL
LIN {X 0,Y 419.136,Z 437.663,A -85,B 0,C 180,E1 -10138.399,E2 -10138.399} C_VEL
LIN {X 0,Y 418.777,Z 447.79,A -85,B 0,C 180,E1 -10141.151,E2 -10141.151} C_VEL
LIN {X 0,Y 418.397,Z 461.213,A -85,B 0,C 180,E1 -10144.638,E2 -10144.638} C_VEL
LIN {X 0,Y 418.101,Z 474.327,A -85,B 0,C 180,E1 -10147.939,E2 -10147.939} C_VEL
LIN {X 0,Y 418.087,Z 476.895,A -85,B 0,C 180,E1 -10148.538,E2 -10148.538} C_VEL
LIN {X 0,Y 420.689,Z 493.121,A -85,B 0,C 180,E1 -10149.231,E2 -10149.231} C_VEL
LIN {X 0,Y 421.754,Z 507.412,A -85,B 0,C 180,E1 -10149.921,E2 -10149.921} C_VEL
LIN {X 0,Y 422.368,Z 521.657,A -85,B 0,C 180,E1 -10150.75,E2 -10150.75} C_VEL
LIN {X 0,Y 422.679,Z 526.479,A -85,B 0,C 180,E1 -10151.08,E2 -10151.08} C_VEL
LIN {X 0,Y 421.64,Z 539.757,A -85,B 0,C 180,E1 -10152.021,E2 -10152.021} C_VEL
LIN {X 0,Y 420.697,Z 551.15,A -85,B 0,C 180,E1 -10153.001,E2 -10153.001} C_VEL
LIN {X 0,Y 419.626,Z 564.106,A -85,B 0,C 180,E1 -10154.331,E2 -10154.331} C_VEL
LIN {X 0,Y 418.888,Z 574.893,A -85,B 0,C 180,E1 -10155.671,E2 -10155.671} C_VEL
LIN {X 0,Y 418.266,Z 585.138,A -85,B 0,C 180,E1 -10157.189,E2 -10157.189} C_VEL
LIN {X 0,Y 417.927,Z 594.434,A -85,B 0,C 180,E1 -10158.848,E2 -10158.848} C_VEL
LIN {X 0,Y 417.693,Z 602.288,A -85,B 0,C 180,E1 -10160.557,E2 -10160.557} C_VEL
LIN {X 0,Y 417.588,Z 608.619,A -85,B 0,C 180,E1 -10162.261,E2 -10162.261} C_VEL
LIN {X 0,Y 417.623,Z 612.397,A -85,B 0,C 180,E1 -10163.498,E2 -10163.498} C_VEL
LIN {X 0,Y 417.734,Z 616.388,A -85,B 0,C 180,E1 -10165.174,E2 -10165.174} C_VEL
LIN {X 0,Y 417.72,Z 618.158,A -85,B 0,C 180,E1 -10166.14,E2 -10166.14} C_VEL
LIN {X 0,Y 417.699,Z 620.54,A -85,B 0,C 180,E1 -10168.071,E2 -10168.071} C_VEL
LIN {X 0,Y 417.859,Z 621.457,A -85,B 0,C 180,E1 -10169.999,E2 -10169.999} C_VEL
LIN {X 0,Y 417.658,Z 620.855,A -85,B 0,C 180,E1 -10171.928,E2 -10171.928} C_VEL
LIN {X 0,Y 417.643,Z 618.81,A -85,B 0,C 180,E1 -10173.858,E2 -10173.858} C_VEL
LIN {X 0,Y 417.536,Z 615.235,A -85,B 0,C 180,E1 -10175.795,E2 -10175.795} C_VEL
LIN {X 0,Y 417.518,Z 611.506,A -85,B 0,C 180,E1 -10177.252,E2 -10177.252} C_VEL
LIN {X 0,Y 417.565,Z 606.816,A -85,B 0,C 180,E1 -10178.711,E2 -10178.711} C_VEL
LIN {X 0,Y 417.73,Z 599.949,A -85,B 0,C 180,E1 -10180.419,E2 -10180.419} C_VEL
LIN {X 0,Y 418.133,Z 591.399,A -85,B 0,C 180,E1 -10182.127,E2 -10182.127} C_VEL
LIN {X 0,Y 418.621,Z 582.49,A -85,B 0,C 180,E1 -10183.593,E2 -10183.593} C_VEL
LIN {X 0,Y 419.379,Z 571.759,A -85,B 0,C 180,E1 -10185.054,E2 -10185.054} C_VEL
LIN {X 0,Y 420.213,Z 560.996,A -85,B 0,C 180,E1 -10186.267,E2 -10186.267} C_VEL
LIN {X 0,Y 421.092,Z 549.349,A -85,B 0,C 180,E1 -10187.356,E2 -10187.356} C_VEL
LIN {X 0,Y 422.118,Z 535.913,A -85,B 0,C 180,E1 -10188.375,E2 -10188.375} C_VEL
LIN {X 0,Y 422.713,Z 523.864,A -85,B 0,C 180,E1 -10189.105,E2 -10189.105} C_VEL
LIN {X 0,Y 421.275,Z 509.485,A -85,B 0,C 180,E1 -10189.849,E2 -10189.849} C_VEL
LIN {X 0,Y 419.203,Z 494.126,A -85,B 0,C 180,E1 -10190.45,E2 -10190.45} C_VEL
LIN {X 0,Y 418.216,Z 487.025,A -85,B 0,C 180,E1 -10190.696,E2 -10190.696} C_VEL
LIN {X 0,Y 418.76,Z 475.596,A -85,B 0,C 180,E1 -10193.751,E2 -10193.751} C_VEL
LIN {X 0,Y 419.412,Z 462.315,A -85,B 0,C 180,E1 -10197.363,E2 -10197.363} C_VEL
LIN {X 0,Y 420.308,Z 448.391,A -85,B 0,C 180,E1 -10201.22,E2 -10201.22} C_VEL
LIN {X 0,Y 421.133,Z 436.63,A -85,B 0,C 180,E1 -10204.568,E2 -10204.568} C_VEL
LIN {X 0,Y 422.379,Z 422.1,A -85,B 0,C 180,E1 -10208.82,E2 -10208.82} C_VEL
LIN {X 0,Y 422.433,Z 418.016,A -85,B 0,C 180,E1 -10210.066,E2 -10210.066} C_VEL
LIN {X 0,Y 421.245,Z 411.234,A -85,B 0,C 180,E1 -10212.281,E2 -10212.281} C_VEL
LIN {X 0,Y 419.06,Z 400.991,A -85,B 0,C 180,E1 -10215.794,E2 -10215.794} C_VEL
LIN {X 0,Y 418.296,Z 397.005,A -85,B 0,C 180,E1 -10217.269,E2 -10217.269} C_VEL
LIN {X 0,Y 418.262,Z 397.009,A -85,B 0,C 180,E1 -10220.615,E2 -10220.615} C_VEL
LIN {X 0,Y 418.238,Z 397.011,A -85,B 0,C 180,E1 -10223.975,E2 -10223.975} C_VEL
LIN {X 0,Y 418.248,Z 397.013,A -85,B 0,C 180,E1 -10227.155,E2 -10227.155} C_VEL
LIN {X 0,Y 418.265,Z 397.009,A -85,B 0,C 180,E1 -10230.838,E2 -10230.838} C_VEL
LIN {X 0,Y 418.261,Z 397.007,A -85,B 0,C 180,E1 -10234.095,E2 -10234.095} C_VEL
LIN {X 0,Y 418.228,Z 397.017,A -85,B 0,C 180,E1 -10237.263,E2 -10237.263} C_VEL
LIN {X 0,Y 418.273,Z 397.007,A -85,B 0,C 180,E1 -10240.364,E2 -10240.364} C_VEL
LIN {X 0,Y 418.306,Z 397.005,A -85,B 0,C 180,E1 -10243.404,E2 -10243.404} C_VEL
LIN {X 0,Y 418.344,Z 397.001,A -85,B 0,C 180,E1 -10246.994,E2 -10246.994} C_VEL
LIN {X 0,Y 418.35,Z 396.997,A -85,B 0,C 180,E1 -10250.329,E2 -10250.329} C_VEL
LIN {X 0,Y 418.483,Z 396.984,A -85,B 0,C 180,E1 -10253.249,E2 -10253.249} C_VEL
LIN {X 0,Y 418.332,Z 397.003,A -85,B 0,C 180,E1 -10255.182,E2 -10255.182} C_VEL
LIN {X 0,Y 418.535,Z 396.974,A -85,B 0,C 180,E1 -10258.076,E2 -10258.076} C_VEL
LIN {X 0,Y 418.664,Z 396.957,A -85,B 0,C 180,E1 -10260,E2 -10260} C_VEL
LIN {X 0,Y 418.502,Z 396.981,A -85,B 0,C 180,E1 -10262.888,E2 -10262.888} C_VEL
LIN {X 0,Y 418.484,Z 396.983,A -85,B 0,C 180,E1 -10266.751,E2 -10266.751} C_VEL
LIN {X 0,Y 418.351,Z 396.996,A -85,B 0,C 180,E1 -10269.671,E2 -10269.671} C_VEL
LIN {X 0,Y 418.346,Z 397.002,A -85,B 0,C 180,E1 -10273.007,E2 -10273.007} C_VEL
LIN {X 0,Y 418.303,Z 397.006,A -85,B 0,C 180,E1 -10276.736,E2 -10276.736} C_VEL
LIN {X 0,Y 418.261,Z 397.007,A -85,B 0,C 180,E1 -10279.791,E2 -10279.791} C_VEL
LIN {X 0,Y 418.229,Z 397.015,A -85,B 0,C 180,E1 -10282.737,E2 -10282.737} C_VEL
LIN {X 0,Y 418.262,Z 397.008,A -85,B 0,C 180,E1 -10285.905,E2 -10285.905} C_VEL
LIN {X 0,Y 418.256,Z 397.01,A -85,B 0,C 180,E1 -10289.163,E2 -10289.163} C_VEL
LIN {X 0,Y 418.25,Z 397.014,A -85,B 0,C 180,E1 -10292.845,E2 -10292.845} C_VEL
LIN {X 0,Y 418.242,Z 397.012,A -85,B 0,C 180,E1 -10296.24,E2 -10296.24} C_VEL
LIN {X 0,Y 418.249,Z 397.009,A -85,B 0,C 180,E1 -10299.683,E2 -10299.683} C_VEL
LIN {X 0,Y 418.227,Z 397.014,A -85,B 0,C 180,E1 -10302.323,E2 -10302.323} C_VEL
LIN {X 0,Y 418.234,Z 397.012,A -85,B 0,C 180,E1 -10305.11,E2 -10305.11} C_VEL
LIN {X 0,Y 418.252,Z 397.009,A -85,B 0,C 180,E1 -10307.77,E2 -10307.77} C_VEL
LIN {X 0,Y 418.265,Z 397.011,A -85,B 0,C 180,E1 -10310.618,E2 -10310.618} C_VEL
LIN {X 0,Y 418.244,Z 397.012,A -85,B 0,C 180,E1 -10313.978,E2 -10313.978} C_VEL
LIN {X 0,Y 418.256,Z 397.009,A -85,B 0,C 180,E1 -10317.157,E2 -10317.157} C_VEL
LIN {X 0,Y 418.267,Z 397.009,A -85,B 0,C 180,E1 -10320.897,E2 -10320.897} C_VEL
LIN {X 0,Y 418.271,Z 397.009,A -85,B 0,C 180,E1 -10324.097,E2 -10324.097} C_VEL
LIN {X 0,Y 418.239,Z 397.01,A -85,B 0,C 180,E1 -10327.265,E2 -10327.265} C_VEL
LIN {X 0,Y 418.285,Z 397.008,A -85,B 0,C 180,E1 -10330.366,E2 -10330.366} C_VEL
LIN {X 0,Y 418.285,Z 397.005,A -85,B 0,C 180,E1 -10333.405,E2 -10333.405} C_VEL
LIN {X 0,Y 418.22,Z 397.189,A -85,B 0,C 180,E1 -10336.014,E2 -10336.014} C_VEL
LIN {X 0,Y 422.307,Z 409.994,A -85,B 0,C 180,E1 -10336.586,E2 -10336.586} C_VEL
LIN {X 0,Y 422.976,Z 412.903,A -85,B 0,C 180,E1 -10336.738,E2 -10336.738} C_VEL
LIN {X 0,Y 422.668,Z 425.175,A -85,B 0,C 180,E1 -10337.356,E2 -10337.356} C_VEL
LIN {X 0,Y 422.234,Z 436.472,A -85,B 0,C 180,E1 -10338.114,E2 -10338.114} C_VEL
LIN {X 0,Y 421.669,Z 447.554,A -85,B 0,C 180,E1 -10339.072,E2 -10339.072} C_VEL
LIN {X 0,Y 421.037,Z 457.573,A -85,B 0,C 180,E1 -10340.15,E2 -10340.15} C_VEL
LIN {X 0,Y 420.431,Z 466.623,A -85,B 0,C 180,E1 -10341.348,E2 -10341.348} C_VEL
LIN {X 0,Y 419.882,Z 475.316,A -85,B 0,C 180,E1 -10342.789,E2 -10342.789} C_VEL
LIN {X 0,Y 419.215,Z 482.355,A -85,B 0,C 180,E1 -10344.228,E2 -10344.228} C_VEL
LIN {X 0,Y 418.935,Z 487.955,A -85,B 0,C 180,E1 -10345.672,E2 -10345.672} C_VEL
LIN {X 0,Y 418.586,Z 492.377,A -85,B 0,C 180,E1 -10347.114,E2 -10347.114} C_VEL
LIN {X 0,Y 418.405,Z 494.708,A -85,B 0,C 180,E1 -10348.076,E2 -10348.076} C_VEL
LIN {X 0,Y 418.163,Z 498.108,A -85,B 0,C 180,E1 -10350.001,E2 -10350.001} C_VEL
LIN {X 0,Y 418.004,Z 499.208,A -85,B 0,C 180,E1 -10350.964,E2 -10350.964} C_VEL
LIN {X 0,Y 418.071,Z 499.871,A -85,B 0,C 180,E1 -10351.928,E2 -10351.928} C_VEL
LIN {X 0,Y 418.002,Z 500.129,A -85,B 0,C 180,E1 -10353.857,E2 -10353.857} C_VEL
LIN {X 0,Y 418.034,Z 499.89,A -85,B 0,C 180,E1 -10354.335,E2 -10354.335} C_VEL
LIN {X 0,Y 417.455,Z 499.512,A -85,B 0,C 180,E1 -10355.139,E2 -10355.139} C_VEL
LIN {X 0,Y 414.765,Z 498.53,A -85,B 0,C 180,E1 -10356.449,E2 -10356.449} C_VEL
LIN {X 0,Y 412.13,Z 496.879,A -85,B 0,C 180,E1 -10357.756,E2 -10357.756} C_VEL
LIN {X 0,Y 411.647,Z 495.318,A -85,B 0,C 180,E1 -10358.548,E2 -10358.548} C_VEL
LIN {X 0,Y 412.026,Z 492.07,A -85,B 0,C 180,E1 -10359.822,E2 -10359.822} C_VEL
LIN {X 0,Y 412.465,Z 487.258,A -85,B 0,C 180,E1 -10361.301,E2 -10361.301} C_VEL
LIN {X 0,Y 412.923,Z 481.174,A -85,B 0,C 180,E1 -10362.784,E2 -10362.784} C_VEL
LIN {X 0,Y 413.447,Z 474.453,A -85,B 0,C 180,E1 -10364.105,E2 -10364.105} C_VEL
LIN {X 0,Y 414.199,Z 465.658,A -85,B 0,C 180,E1 -10365.501,E2 -10365.501} C_VEL
LIN {X 0,Y 414.897,Z 456.076,A -85,B 0,C 180,E1 -10366.737,E2 -10366.737} C_VEL
LIN {X 0,Y 415.591,Z 445.242,A -85,B 0,C 180,E1 -10367.85,E2 -10367.85} C_VEL
LIN {X 0,Y 416.131,Z 434.652,A -85,B 0,C 180,E1 -10368.718,E2 -10368.718} C_VEL
LIN {X 0,Y 416.686,Z 423.111,A -85,B 0,C 180,E1 -10369.452,E2 -10369.452} C_VEL
LIN {X 0,Y 416.732,Z 414.391,A -85,B 0,C 180,E1 -10369.89,E2 -10369.89} C_VEL
LIN {X 0,Y 412.435,Z 401.89,A -85,B 0,C 180,E1 -10370.567,E2 -10370.567} C_VEL
LIN {X 0,Y 411.104,Z 397.904,A -85,B 0,C 180,E1 -10370.738,E2 -10370.738} C_VEL
LIN {X 0,Y 411.199,Z 397.89,A -85,B 0,C 180,E1 -10373.149,E2 -10373.149} C_VEL
LIN {X 0,Y 411.244,Z 397.883,A -85,B 0,C 180,E1 -10376.381,E2 -10376.381} C_VEL
LIN {X 0,Y 411.207,Z 397.889,A -85,B 0,C 180,E1 -10379.713,E2 -10379.713} C_VEL
LIN {X 0,Y 411.212,Z 397.891,A -85,B 0,C 180,E1 -10383.156,E2 -10383.156} C_VEL
LIN {X 0,Y 411.198,Z 397.891,A -85,B 0,C 180,E1 -10386.553,E2 -10386.553} C_VEL
LIN {X 0,Y 411.217,Z 397.882,A -85,B 0,C 180,E1 -10389.728,E2 -10389.728} C_VEL
LIN {X 0,Y 411.179,Z 397.89,A -85,B 0,C 180,E1 -10393.134,E2 -10393.134} C_VEL
LIN {X 0,Y 411.178,Z 397.888,A -85,B 0,C 180,E1 -10395.88,E2 -10395.88} C_VEL
LIN {X 0,Y 411.173,Z 397.887,A -85,B 0,C 180,E1 -10398.771,E2 -10398.771} C_VEL
LIN {X 0,Y 411.204,Z 397.868,A -85,B 0,C 180,E1 -10402.027,E2 -10402.027} C_VEL
LIN {X 0,Y 411.212,Z 397.888,A -85,B 0,C 180,E1 -10405.667,E2 -10405.667} C_VEL
LIN {X 0,Y 411.194,Z 397.871,A -85,B 0,C 180,E1 -10409.152,E2 -10409.152} C_VEL
LIN {X 0,Y 411.264,Z 397.87,A -85,B 0,C 180,E1 -10412.522,E2 -10412.522} C_VEL
LIN {X 0,Y 411.224,Z 397.889,A -85,B 0,C 180,E1 -10415.784,E2 -10415.784} C_VEL
LIN {X 0,Y 411.201,Z 397.888,A -85,B 0,C 180,E1 -10418.966,E2 -10418.966} C_VEL
LIN {X 0,Y 411.242,Z 397.898,A -85,B 0,C 180,E1 -10421.359,E2 -10421.359} C_VEL
LIN {X 0,Y 414.942,Z 410.132,A -85,B 0,C 180,E1 -10422.249,E2 -10422.249} C_VEL
LIN {X 0,Y 416.642,Z 416.703,A -85,B 0,C 180,E1 -10422.786,E2 -10422.786} C_VEL
LIN {X 0,Y 415.9,Z 429.538,A -85,B 0,C 180,E1 -10423.81,E2 -10423.81} C_VEL
LIN {X 0,Y 415.069,Z 441.997,A -85,B 0,C 180,E1 -10425.03,E2 -10425.03} C_VEL
LIN {X 0,Y 414.267,Z 452.367,A -85,B 0,C 180,E1 -10426.26,E2 -10426.26} C_VEL
LIN {X 0,Y 413.413,Z 462.685,A -85,B 0,C 180,E1 -10427.731,E2 -10427.731} C_VEL
LIN {X 0,Y 412.876,Z 471.247,A -85,B 0,C 180,E1 -10429.208,E2 -10429.208} C_VEL
LIN {X 0,Y 412.251,Z 479.469,A -85,B 0,C 180,E1 -10430.927,E2 -10430.927} C_VEL
LIN {X 0,Y 411.8,Z 486.122,A -85,B 0,C 180,E1 -10432.646,E2 -10432.646} C_VEL
LIN {X 0,Y 411.46,Z 492.065,A -85,B 0,C 180,E1 -10434.609,E2 -10434.609} C_VEL
LIN {X 0,Y 411.119,Z 495.485,A -85,B 0,C 180,E1 -10436.079,E2 -10436.079} C_VEL
LIN {X 0,Y 411.057,Z 498.733,A -85,B 0,C 180,E1 -10438.04,E2 -10438.04} C_VEL
LIN {X 0,Y 411.042,Z 500.621,A -85,B 0,C 180,E1 -10440,E2 -10440} C_VEL
LIN {X 0,Y 411.168,Z 501.169,A -85,B 0,C 180,E1 -10441.959,E2 -10441.959} C_VEL
LIN {X 0,Y 411.233,Z 500.414,A -85,B 0,C 180,E1 -10443.92,E2 -10443.92} C_VEL
LIN {X 0,Y 411.535,Z 498.265,A -85,B 0,C 180,E1 -10445.881,E2 -10445.881} C_VEL
LIN {X 0,Y 412.035,Z 494.665,A -85,B 0,C 180,E1 -10447.843,E2 -10447.843} C_VEL
LIN {X 0,Y 412.615,Z 489.555,A -85,B 0,C 180,E1 -10449.807,E2 -10449.807} C_VEL
LIN {X 0,Y 413.153,Z 484.646,A -85,B 0,C 180,E1 -10451.281,E2 -10451.281} C_VEL
LIN {X 0,Y 413.952,Z 477.525,A -85,B 0,C 180,E1 -10453,E2 -10453} C_VEL
LIN {X 0,Y 414.99,Z 468.655,A -85,B 0,C 180,E1 -10454.716,E2 -10454.716} C_VEL
LIN {X 0,Y 416.041,Z 459.305,A -85,B 0,C 180,E1 -10456.184,E2 -10456.184} C_VEL
LIN {X 0,Y 417.002,Z 448.992,A -85,B 0,C 180,E1 -10457.533,E2 -10457.533} C_VEL
LIN {X 0,Y 418.056,Z 437.582,A -85,B 0,C 180,E1 -10458.754,E2 -10458.754} C_VEL
LIN {X 0,Y 418.978,Z 426.074,A -85,B 0,C 180,E1 -10459.765,E2 -10459.765} C_VEL
LIN {X 0,Y 419.428,Z 419.954,A -85,B 0,C 180,E1 -10460.224,E2 -10460.224} C_VEL
LIN {X 0,Y 417.078,Z 412.238,A -85,B 0,C 180,E1 -10460.97,E2 -10460.97} C_VEL
LIN {X 0,Y 412.535,Z 401.2,A -85,B 0,C 180,E1 -10462.011,E2 -10462.011} C_VEL
LIN {X 0,Y 411.278,Z 398.263,A -85,B 0,C 180,E1 -10462.267,E2 -10462.267} C_VEL
LIN {X 0,Y 411.204,Z 397.894,A -85,B 0,C 180,E1 -10462.334,E2 -10462.334} C_VEL
LIN {X 0,Y 411.24,Z 397.889,A -85,B 0,C 180,E1 -10465.293,E2 -10465.293} C_VEL
LIN {X 0,Y 411.262,Z 397.883,A -85,B 0,C 180,E1 -10467.477,E2 -10467.477} C_VEL
LIN {X 0,Y 411.193,Z 397.892,A -85,B 0,C 180,E1 -10470.847,E2 -10470.847} C_VEL
LIN {X 0,Y 411.209,Z 397.891,A -85,B 0,C 180,E1 -10474.333,E2 -10474.333} C_VEL
LIN {X 0,Y 411.197,Z 397.891,A -85,B 0,C 180,E1 -10477.973,E2 -10477.973} C_VEL
LIN {X 0,Y 411.184,Z 397.893,A -85,B 0,C 180,E1 -10480.504,E2 -10480.504} C_VEL
LIN {X 0,Y 411.182,Z 398.055,A -85,B 0,C 180,E1 -10483.132,E2 -10483.132} C_VEL
LIN {X 0,Y 412.209,Z 402.675,A -85,B 0,C 180,E1 -10485.732,E2 -10485.732} C_VEL
LIN {X 0,Y 413.415,Z 408.537,A -85,B 0,C 180,E1 -10488.47,E2 -10488.47} C_VEL
LIN {X 0,Y 414.199,Z 413.558,A -85,B 0,C 180,E1 -10490.484,E2 -10490.484} C_VEL
LIN {X 0,Y 413.799,Z 417.385,A -85,B 0,C 180,E1 -10491.808,E2 -10491.808} C_VEL
LIN {X 0,Y 412.579,Z 430.006,A -85,B 0,C 180,E1 -10495.796,E2 -10495.796} C_VEL
LIN {X 0,Y 412.003,Z 441.823,A -85,B 0,C 180,E1 -10499.219,E2 -10499.219} C_VEL
LIN {X 0,Y 411.55,Z 453.997,A -85,B 0,C 180,E1 -10502.543,E2 -10502.543} C_VEL
LIN {X 0,Y 411.185,Z 466.353,A -85,B 0,C 180,E1 -10505.781,E2 -10505.781} C_VEL
LIN {X 0,Y 411.018,Z 475.111,A -85,B 0,C 180,E1 -10508.001,E2 -10508.001} C_VEL
LIN {X 0,Y 413.857,Z 492.006,A -85,B 0,C 180,E1 -10508.775,E2 -10508.775} C_VEL
LIN {X 0,Y 414.968,Z 505.396,A -85,B 0,C 180,E1 -10509.458,E2 -10509.458} C_VEL
LIN {X 0,Y 415.46,Z 520.453,A -85,B 0,C 180,E1 -10510.353,E2 -10510.353} C_VEL
LIN {X 0,Y 415.784,Z 527.947,A -85,B 0,C 180,E1 -10510.882,E2 -10510.882} C_VEL
LIN {X 0,Y 414.636,Z 541.366,A -85,B 0,C 180,E1 -10511.901,E2 -10511.901} C_VEL
LIN {X 0,Y 413.615,Z 552.891,A -85,B 0,C 180,E1 -10512.955,E2 -10512.955} C_VEL
LIN {X 0,Y 412.531,Z 565.254,A -85,B 0,C 180,E1 -10514.308,E2 -10514.308} C_VEL
LIN {X 0,Y 411.807,Z 575.67,A -85,B 0,C 180,E1 -10515.672,E2 -10515.672} C_VEL
LIN {X 0,Y 411.178,Z 585.273,A -85,B 0,C 180,E1 -10517.161,E2 -10517.161} C_VEL
LIN {X 0,Y 410.845,Z 594.632,A -85,B 0,C 180,E1 -10518.904,E2 -10518.904} C_VEL
LIN {X 0,Y 410.6,Z 602.254,A -85,B 0,C 180,E1 -10520.641,E2 -10520.641} C_VEL
LIN {X 0,Y 410.532,Z 607.565,A -85,B 0,C 180,E1 -10522.127,E2 -10522.127} C_VEL
LIN {X 0,Y 410.578,Z 611.541,A -85,B 0,C 180,E1 -10523.463,E2 -10523.463} C_VEL
LIN {X 0,Y 410.687,Z 615.344,A -85,B 0,C 180,E1 -10525.091,E2 -10525.091} C_VEL
LIN {X 0,Y 410.684,Z 617.112,A -85,B 0,C 180,E1 -10526.074,E2 -10526.074} C_VEL
LIN {X 0,Y 410.668,Z 619.487,A -85,B 0,C 180,E1 -10528.038,E2 -10528.038} C_VEL
LIN {X 0,Y 410.771,Z 620.132,A -85,B 0,C 180,E1 -10529.019,E2 -10529.019} C_VEL
LIN {X 0,Y 410.839,Z 620.404,A -85,B 0,C 180,E1 -10529.999,E2 -10529.999} C_VEL
LIN {X 0,Y 410.629,Z 619.792,A -85,B 0,C 180,E1 -10531.961,E2 -10531.961} C_VEL
LIN {X 0,Y 410.606,Z 617.731,A -85,B 0,C 180,E1 -10533.925,E2 -10533.925} C_VEL
LIN {X 0,Y 410.487,Z 614.13,A -85,B 0,C 180,E1 -10535.895,E2 -10535.895} C_VEL
LIN {X 0,Y 410.47,Z 610.369,A -85,B 0,C 180,E1 -10537.377,E2 -10537.377} C_VEL
LIN {X 0,Y 410.489,Z 605.642,A -85,B 0,C 180,E1 -10538.863,E2 -10538.863} C_VEL
LIN {X 0,Y 410.696,Z 598.725,A -85,B 0,C 180,E1 -10540.599,E2 -10540.599} C_VEL
LIN {X 0,Y 411.03,Z 591.495,A -85,B 0,C 180,E1 -10542.089,E2 -10542.089} C_VEL
LIN {X 0,Y 411.517,Z 582.701,A -85,B 0,C 180,E1 -10543.594,E2 -10543.594} C_VEL
LIN {X 0,Y 412.28,Z 572.301,A -85,B 0,C 180,E1 -10545.066,E2 -10545.066} C_VEL
LIN {X 0,Y 413.222,Z 560.665,A -85,B 0,C 180,E1 -10546.423,E2 -10546.423} C_VEL
LIN {X 0,Y 414.115,Z 549.148,A -85,B 0,C 180,E1 -10547.531,E2 -10547.531} C_VEL
LIN {X 0,Y 415.159,Z 535.987,A -85,B 0,C 180,E1 -10548.56,E2 -10548.56} C_VEL
LIN {X 0,Y 415.824,Z 525.191,A -85,B 0,C 180,E1 -10549.242,E2 -10549.242} C_VEL
LIN {X 0,Y 414.414,Z 510.634,A -85,B 0,C 180,E1 -10550.042,E2 -10550.042} C_VEL
LIN {X 0,Y 412.528,Z 495.908,A -85,B 0,C 180,E1 -10550.669,E2 -10550.669} C_VEL
LIN {X 0,Y 411.202,Z 486.291,A -85,B 0,C 180,E1 -10550.983,E2 -10550.983} C_VEL
LIN {X 0,Y 411.73,Z 474.59,A -85,B 0,C 180,E1 -10554.182,E2 -10554.182} C_VEL
LIN {X 0,Y 412.412,Z 462.229,A -85,B 0,C 180,E1 -10557.608,E2 -10557.608} C_VEL
LIN {X 0,Y 413.272,Z 449.423,A -85,B 0,C 180,E1 -10561.23,E2 -10561.23} C_VEL
LIN {X 0,Y 414.125,Z 437.629,A -85,B 0,C 180,E1 -10564.645,E2 -10564.645} C_VEL
LIN {X 0,Y 415.406,Z 423.337,A -85,B 0,C 180,E1 -10568.9,E2 -10568.9} C_VEL
LIN {X 0,Y 415.357,Z 418.529,A -85,B 0,C 180,E1 -10570.411,E2 -10570.411} C_VEL
LIN {X 0,Y 414.017,Z 411.474,A -85,B 0,C 180,E1 -10572.764,E2 -10572.764} C_VEL
LIN {X 0,Y 411.899,Z 401.311,A -85,B 0,C 180,E1 -10576.322,E2 -10576.322} C_VEL
LIN {X 0,Y 411.246,Z 397.885,A -85,B 0,C 180,E1 -10577.638,E2 -10577.638} C_VEL
LIN {X 0,Y 411.225,Z 397.886,A -85,B 0,C 180,E1 -10580.777,E2 -10580.777} C_VEL
LIN {X 0,Y 411.191,Z 397.888,A -85,B 0,C 180,E1 -10584.471,E2 -10584.471} C_VEL
LIN {X 0,Y 411.198,Z 397.89,A -85,B 0,C 180,E1 -10586.873,E2 -10586.873} C_VEL
LIN {X 0,Y 411.231,Z 397.885,A -85,B 0,C 180,E1 -10590.641,E2 -10590.641} C_VEL
LIN {X 0,Y 411.228,Z 397.885,A -85,B 0,C 180,E1 -10593.619,E2 -10593.619} C_VEL
LIN {X 0,Y 411.193,Z 397.89,A -85,B 0,C 180,E1 -10596.852,E2 -10596.852} C_VEL
LIN {X 0,Y 411.204,Z 397.886,A -85,B 0,C 180,E1 -10600.05,E2 -10600.05} C_VEL
LIN {X 0,Y 411.252,Z 397.885,A -85,B 0,C 180,E1 -10603.131,E2 -10603.131} C_VEL
LIN {X 0,Y 411.303,Z 397.877,A -85,B 0,C 180,E1 -10606.891,E2 -10606.891} C_VEL
LIN {X 0,Y 411.298,Z 397.875,A -85,B 0,C 180,E1 -10610.162,E2 -10610.162} C_VEL
LIN {X 0,Y 411.45,Z 397.861,A -85,B 0,C 180,E1 -10613.133,E2 -10613.133} C_VEL
LIN {X 0,Y 411.303,Z 397.879,A -85,B 0,C 180,E1 -10615.099,E2 -10615.099} C_VEL
LIN {X 0,Y 411.504,Z 397.849,A -85,B 0,C 180,E1 -10618.043,E2 -10618.043} C_VEL
LIN {X 0,Y 411.633,Z 397.833,A -85,B 0,C 180,E1 -10620,E2 -10620} C_VEL
LIN {X 0,Y 411.458,Z 397.859,A -85,B 0,C 180,E1 -10622.938,E2 -10622.938} C_VEL
LIN {X 0,Y 411.451,Z 397.86,A -85,B 0,C 180,E1 -10626.867,E2 -10626.867} C_VEL
LIN {X 0,Y 411.299,Z 397.874,A -85,B 0,C 180,E1 -10629.839,E2 -10629.839} C_VEL
LIN {X 0,Y 411.304,Z 397.877,A -85,B 0,C 180,E1 -10633.11,E2 -10633.11} C_VEL
LIN {X 0,Y 411.247,Z 397.886,A -85,B 0,C 180,E1 -10636.889,E2 -10636.889} C_VEL
LIN {X 0,Y 411.221,Z 397.885,A -85,B 0,C 180,E1 -10639.988,E2 -10639.988} C_VEL
LIN {X 0,Y 411.194,Z 397.89,A -85,B 0,C 180,E1 -10643.148,E2 -10643.148} C_VEL
LIN {X 0,Y 411.229,Z 397.886,A -85,B 0,C 180,E1 -10646.382,E2 -10646.382} C_VEL
LIN {X 0,Y 411.192,Z 397.888,A -85,B 0,C 180,E1 -10649.714,E2 -10649.714} C_VEL
LIN {X 0,Y 411.199,Z 397.889,A -85,B 0,C 180,E1 -10653.157,E2 -10653.157} C_VEL
LIN {X 0,Y 411.189,Z 397.892,A -85,B 0,C 180,E1 -10656.554,E2 -10656.554} C_VEL
LIN {X 0,Y 411.213,Z 397.885,A -85,B 0,C 180,E1 -10659.73,E2 -10659.73} C_VEL
LIN {X 0,Y 411.173,Z 397.891,A -85,B 0,C 180,E1 -10663.134,E2 -10663.134} C_VEL
LIN {X 0,Y 411.164,Z 397.892,A -85,B 0,C 180,E1 -10665.882,E2 -10665.882} C_VEL
LIN {X 0,Y 411.197,Z 397.891,A -85,B 0,C 180,E1 -10668.767,E2 -10668.767} C_VEL
LIN {X 0,Y 411.202,Z 397.889,A -85,B 0,C 180,E1 -10672.029,E2 -10672.029} C_VEL
LIN {X 0,Y 411.204,Z 397.887,A -85,B 0,C 180,E1 -10675.668,E2 -10675.668} C_VEL
LIN {X 0,Y 411.188,Z 397.889,A -85,B 0,C 180,E1 -10679.154,E2 -10679.154} C_VEL
LIN {X 0,Y 411.258,Z 397.884,A -85,B 0,C 180,E1 -10682.524,E2 -10682.524} C_VEL
LIN {X 0,Y 411.227,Z 397.885,A -85,B 0,C 180,E1 -10685.786,E2 -10685.786} C_VEL
LIN {X 0,Y 411.197,Z 397.888,A -85,B 0,C 180,E1 -10688.967,E2 -10688.967} C_VEL
LIN {X 0,Y 411.25,Z 397.884,A -85,B 0,C 180,E1 -10692.086,E2 -10692.086} C_VEL
LIN {X 0,Y 411.154,Z 397.895,A -85,B 0,C 180,E1 -10695.145,E2 -10695.145} C_VEL
LIN {X 0,Y 411.145,Z 397.899,A -85,B 0,C 180,E1 -10695.718,E2 -10695.718} C_VEL
LIN {X 0,Y 415.45,Z 411.393,A -85,B 0,C 180,E1 -10696.342,E2 -10696.342} C_VEL
LIN {X 0,Y 416.191,Z 414.696,A -85,B 0,C 180,E1 -10696.52,E2 -10696.52} C_VEL
LIN {X 0,Y 415.851,Z 426.741,A -85,B 0,C 180,E1 -10697.146,E2 -10697.146} C_VEL
LIN {X 0,Y 415.381,Z 437.874,A -85,B 0,C 180,E1 -10697.915,E2 -10697.915} C_VEL
LIN {X 0,Y 414.812,Z 448.879,A -85,B 0,C 180,E1 -10698.89,E2 -10698.89} C_VEL
LIN {X 0,Y 414.09,Z 459.727,A -85,B 0,C 180,E1 -10700.09,E2 -10700.09} C_VEL
LIN {X 0,Y 413.353,Z 469.405,A -85,B 0,C 180,E1 -10701.445,E2 -10701.445} C_VEL
LIN {X 0,Y 412.807,Z 477.792,A -85,B 0,C 180,E1 -10702.911,E2 -10702.911} C_VEL
LIN {X 0,Y 412.243,Z 483.503,A -85,B 0,C 180,E1 -10704.13,E2 -10704.13} C_VEL
LIN {X 0,Y 411.945,Z 489.076,A -85,B 0,C 180,E1 -10705.598,E2 -10705.598} C_VEL
LIN {X 0,Y 411.582,Z 493.469,A -85,B 0,C 180,E1 -10707.065,E2 -10707.065} C_VEL
LIN {X 0,Y 411.393,Z 495.78,A -85,B 0,C 180,E1 -10708.043,E2 -10708.043} C_VEL
LIN {X 0,Y 411.145,Z 499.159,A -85,B 0,C 180,E1 -10710.001,E2 -10710.001} C_VEL
LIN {X 0,Y 410.981,Z 500.238,A -85,B 0,C 180,E1 -10710.981,E2 -10710.981} C_VEL
LIN {X 0,Y 411.048,Z 500.89,A -85,B 0,C 180,E1 -10711.961,E2 -10711.961} C_VEL
LIN {X 0,Y 410.916,Z 501.207,A -85,B 0,C 180,E1 -10712.942,E2 -10712.942} C_VEL
LIN {X 0,Y 411.011,Z 500.904,A -85,B 0,C 180,E1 -10714.358,E2 -10714.358} C_VEL
LIN {X 0,Y 411.3,Z 499.724,A -85,B 0,C 180,E1 -10715.886,E2 -10715.886} C_VEL
LIN {X 0,Y 411.356,Z 498.473,A -85,B 0,C 180,E1 -10716.87,E2 -10716.87} C_VEL
LIN {X 0,Y 411.647,Z 495.318,A -85,B 0,C 180,E1 -10718.548,E2 -10718.548} C_VEL
LIN {X 0,Y 411.201,Z 493.568,A -85,B 0,C 180,E1 -10719.33,E2 -10719.33} C_VEL
LIN {X 0,Y 408.759,Z 490.415,A -85,B 0,C 180,E1 -10720.602,E2 -10720.602} C_VEL
LIN {X 0,Y 406.696,Z 487.503,A -85,B 0,C 180,E1 -10721.601,E2 -10721.601} C_VEL
LIN {X 0,Y 405.91,Z 484.86,A -85,B 0,C 180,E1 -10722.34,E2 -10722.34} C_VEL
LIN {X 0,Y 405.904,Z 483.853,A -85,B 0,C 180,E1 -10722.581,E2 -10722.581} C_VEL
LIN {X 0,Y 406.411,Z 477.082,A -85,B 0,C 180,E1 -10724.011,E2 -10724.011} C_VEL
LIN {X 0,Y 407.151,Z 469.771,A -85,B 0,C 180,E1 -10725.263,E2 -10725.263} C_VEL
LIN {X 0,Y 407.878,Z 460.9,A -85,B 0,C 180,E1 -10726.518,E2 -10726.518} C_VEL
LIN {X 0,Y 408.536,Z 451.021,A -85,B 0,C 180,E1 -10727.651,E2 -10727.651} C_VEL
LIN {X 0,Y 409.189,Z 440.075,A -85,B 0,C 180,E1 -10728.657,E2 -10728.657} C_VEL
LIN {X 0,Y 409.76,Z 429.209,A -85,B 0,C 180,E1 -10729.442,E2 -10729.442} C_VEL
LIN {X 0,Y 410.158,Z 417.163,A -85,B 0,C 180,E1 -10730.104,E2 -10730.104} C_VEL
LIN {X 0,Y 409.175,Z 413.346,A -85,B 0,C 180,E1 -10730.331,E2 -10730.331} C_VEL
LIN {X 0,Y 404.747,Z 401.09,A -85,B 0,C 180,E1 -10730.983,E2 -10730.983} C_VEL
LIN {X 0,Y 404.07,Z 398.78,A -85,B 0,C 180,E1 -10731.093,E2 -10731.093} C_VEL
LIN {X 0,Y 404.167,Z 398.764,A -85,B 0,C 180,E1 -10733.576,E2 -10733.576} C_VEL
LIN {X 0,Y 404.19,Z 398.761,A -85,B 0,C 180,E1 -10735.767,E2 -10735.767} C_VEL
LIN {X 0,Y 404.201,Z 398.759,A -85,B 0,C 180,E1 -10738,E2 -10738} C_VEL
LIN {X 0,Y 404.145,Z 398.769,A -85,B 0,C 180,E1 -10741.558,E2 -10741.558} C_VEL
LIN {X 0,Y 404.189,Z 398.766,A -85,B 0,C 180,E1 -10745.017,E2 -10745.017} C_VEL
LIN {X 0,Y 404.158,Z 398.758,A -85,B 0,C 180,E1 -10748.757,E2 -10748.757} C_VEL
LIN {X 0,Y 404.128,Z 398.768,A -85,B 0,C 180,E1 -10751.6,E2 -10751.6} C_VEL
LIN {X 0,Y 404.152,Z 398.767,A -85,B 0,C 180,E1 -10754.522,E2 -10754.522} C_VEL
LIN {X 0,Y 404.179,Z 398.761,A -85,B 0,C 180,E1 -10757.301,E2 -10757.301} C_VEL
LIN {X 0,Y 404.174,Z 398.75,A -85,B 0,C 180,E1 -10759.955,E2 -10759.955} C_VEL
LIN {X 0,Y 404.145,Z 398.758,A -85,B 0,C 180,E1 -10763.124,E2 -10763.124} C_VEL
LIN {X 0,Y 404.15,Z 398.767,A -85,B 0,C 180,E1 -10766.188,E2 -10766.188} C_VEL
LIN {X 0,Y 404.15,Z 398.739,A -85,B 0,C 180,E1 -10769.715,E2 -10769.715} C_VEL
LIN {X 0,Y 404.199,Z 398.75,A -85,B 0,C 180,E1 -10773.123,E2 -10773.123} C_VEL
LIN {X 0,Y 404.178,Z 398.763,A -85,B 0,C 180,E1 -10775.334,E2 -10775.334} C_VEL
LIN {X 0,Y 404.143,Z 398.766,A -85,B 0,C 180,E1 -10778.58,E2 -10778.58} C_VEL
LIN {X 0,Y 404.188,Z 398.764,A -85,B 0,C 180,E1 -10781.088,E2 -10781.088} C_VEL
LIN {X 0,Y 408.268,Z 412.305,A -85,B 0,C 180,E1 -10782.096,E2 -10782.096} C_VEL
LIN {X 0,Y 409.767,Z 417.531,A -85,B 0,C 180,E1 -10782.538,E2 -10782.538} C_VEL
LIN {X 0,Y 408.99,Z 431.231,A -85,B 0,C 180,E1 -10783.657,E2 -10783.657} C_VEL
LIN {X 0,Y 408.138,Z 443.566,A -85,B 0,C 180,E1 -10784.9,E2 -10784.9} C_VEL
LIN {X 0,Y 407.224,Z 454.721,A -85,B 0,C 180,E1 -10786.272,E2 -10786.272} C_VEL
LIN {X 0,Y 406.392,Z 464.794,A -85,B 0,C 180,E1 -10787.769,E2 -10787.769} C_VEL
LIN {X 0,Y 405.72,Z 474.447,A -85,B 0,C 180,E1 -10789.52,E2 -10789.52} C_VEL
LIN {X 0,Y 405.21,Z 481.254,A -85,B 0,C 180,E1 -10791.019,E2 -10791.019} C_VEL
LIN {X 0,Y 404.819,Z 486.929,A -85,B 0,C 180,E1 -10792.518,E2 -10792.518} C_VEL
LIN {X 0,Y 404.466,Z 492.931,A -85,B 0,C 180,E1 -10794.516,E2 -10794.516} C_VEL
LIN {X 0,Y 404.098,Z 496.414,A -85,B 0,C 180,E1 -10796.011,E2 -10796.011} C_VEL
LIN {X 0,Y 404.037,Z 499.722,A -85,B 0,C 180,E1 -10798.006,E2 -10798.006} C_VEL
LIN {X 0,Y 404.033,Z 501.672,A -85,B 0,C 180,E1 -10800,E2 -10800} C_VEL
LIN {X 0,Y 404.168,Z 502.274,A -85,B 0,C 180,E1 -10801.993,E2 -10801.993} C_VEL
LIN {X 0,Y 404.262,Z 501.564,A -85,B 0,C 180,E1 -10803.987,E2 -10803.987} C_VEL
LIN {X 0,Y 404.573,Z 499.469,A -85,B 0,C 180,E1 -10805.982,E2 -10805.982} C_VEL
LIN {X 0,Y 405.122,Z 495.941,A -85,B 0,C 180,E1 -10807.977,E2 -10807.977} C_VEL
LIN {X 0,Y 405.759,Z 490.907,A -85,B 0,C 180,E1 -10809.974,E2 -10809.974} C_VEL
LIN {X 0,Y 406.325,Z 486.044,A -85,B 0,C 180,E1 -10811.473,E2 -10811.473} C_VEL
LIN {X 0,Y 407.203,Z 478.967,A -85,B 0,C 180,E1 -10813.219,E2 -10813.219} C_VEL
LIN {X 0,Y 408.302,Z 470.199,A -85,B 0,C 180,E1 -10814.963,E2 -10814.963} C_VEL
LIN {X 0,Y 409.428,Z 461.011,A -85,B 0,C 180,E1 -10816.453,E2 -10816.453} C_VEL
LIN {X 0,Y 410.471,Z 450.818,A -85,B 0,C 180,E1 -10817.821,E2 -10817.821} C_VEL
LIN {X 0,Y 411.558,Z 439.535,A -85,B 0,C 180,E1 -10819.062,E2 -10819.062} C_VEL
LIN {X 0,Y 412.596,Z 427.896,A -85,B 0,C 180,E1 -10820.119,E2 -10820.119} C_VEL
LIN {X 0,Y 413.004,Z 421.531,A -85,B 0,C 180,E1 -10820.621,E2 -10820.621} C_VEL
LIN {X 0,Y 409.296,Z 410.746,A -85,B 0,C 180,E1 -10821.714,E2 -10821.714} C_VEL
LIN {X 0,Y 404.605,Z 400.509,A -85,B 0,C 180,E1 -10822.752,E2 -10822.752} C_VEL
LIN {X 0,Y 404.177,Z 398.772,A -85,B 0,C 180,E1 -10822.91,E2 -10822.91} C_VEL
LIN {X 0,Y 404.187,Z 398.767,A -85,B 0,C 180,E1 -10825.766,E2 -10825.766} C_VEL
LIN {X 0,Y 404.198,Z 398.763,A -85,B 0,C 180,E1 -10827.999,E2 -10827.999} C_VEL
LIN {X 0,Y 404.142,Z 398.769,A -85,B 0,C 180,E1 -10831.558,E2 -10831.558} C_VEL
LIN {X 0,Y 404.187,Z 398.763,A -85,B 0,C 180,E1 -10835.016,E2 -10835.016} C_VEL
LIN {X 0,Y 404.158,Z 398.769,A -85,B 0,C 180,E1 -10838.756,E2 -10838.756} C_VEL
LIN {X 0,Y 404.139,Z 398.771,A -85,B 0,C 180,E1 -10842.237,E2 -10842.237} C_VEL
LIN {X 0,Y 405.245,Z 403.917,A -85,B 0,C 180,E1 -10845.32,E2 -10845.32} C_VEL
LIN {X 0,Y 406.402,Z 409.497,A -85,B 0,C 180,E1 -10848.04,E2 -10848.04} C_VEL
LIN {X 0,Y 407.286,Z 414.973,A -85,B 0,C 180,E1 -10850.322,E2 -10850.322} C_VEL
LIN {X 0,Y 406.979,Z 418.422,A -85,B 0,C 180,E1 -10851.561,E2 -10851.561} C_VEL
LIN {X 0,Y 405.604,Z 431.253,A -85,B 0,C 180,E1 -10855.727,E2 -10855.727} C_VEL
LIN {X 0,Y 404.982,Z 442.966,A -85,B 0,C 180,E1 -10859.206,E2 -10859.206} C_VEL
LIN {X 0,Y 404.519,Z 454.33,A -85,B 0,C 180,E1 -10862.382,E2 -10862.382} C_VEL
LIN {X 0,Y 404.133,Z 467.369,A -85,B 0,C 180,E1 -10865.878,E2 -10865.878} C_VEL
LIN {X 0,Y 403.993,Z 473.482,A -85,B 0,C 180,E1 -10867.429,E2 -10867.429} C_VEL
LIN {X 0,Y 407.044,Z 490.578,A -85,B 0,C 180,E1 -10868.275,E2 -10868.275} C_VEL
LIN {X 0,Y 408.254,Z 504.295,A -85,B 0,C 180,E1 -10869.011,E2 -10869.011} C_VEL
LIN {X 0,Y 408.669,Z 520.367,A -85,B 0,C 180,E1 -10870.013,E2 -10870.013} C_VEL
LIN {X 0,Y 408.895,Z 529.375,A -85,B 0,C 180,E1 -10870.678,E2 -10870.678} C_VEL
LIN {X 0,Y 407.629,Z 543,A -85,B 0,C 180,E1 -10871.777,E2 -10871.777} C_VEL
LIN {X 0,Y 406.444,Z 555.789,A -85,B 0,C 180,E1 -10873.034,E2 -10873.034} C_VEL
LIN {X 0,Y 405.388,Z 567.421,A -85,B 0,C 180,E1 -10874.411,E2 -10874.411} C_VEL
LIN {X 0,Y 404.599,Z 578.122,A -85,B 0,C 180,E1 -10875.925,E2 -10875.925} C_VEL
LIN {X 0,Y 403.977,Z 588.512,A -85,B 0,C 180,E1 -10877.694,E2 -10877.694} C_VEL
LIN {X 0,Y 403.621,Z 597.056,A -85,B 0,C 180,E1 -10879.464,E2 -10879.464} C_VEL
LIN {X 0,Y 403.495,Z 603.084,A -85,B 0,C 180,E1 -10880.98,E2 -10880.98} C_VEL
LIN {X 0,Y 403.479,Z 609.535,A -85,B 0,C 180,E1 -10882.996,E2 -10882.996} C_VEL
LIN {X 0,Y 403.64,Z 614.304,A -85,B 0,C 180,E1 -10885.005,E2 -10885.005} C_VEL
LIN {X 0,Y 403.649,Z 616.066,A -85,B 0,C 180,E1 -10886.005,E2 -10886.005} C_VEL
LIN {X 0,Y 403.637,Z 618.433,A -85,B 0,C 180,E1 -10888.003,E2 -10888.003} C_VEL
LIN {X 0,Y 403.759,Z 619.078,A -85,B 0,C 180,E1 -10889.002,E2 -10889.002} C_VEL
LIN {X 0,Y 403.82,Z 619.345,A -85,B 0,C 180,E1 -10889.999,E2 -10889.999} C_VEL
LIN {X 0,Y 403.601,Z 618.72,A -85,B 0,C 180,E1 -10891.995,E2 -10891.995} C_VEL
LIN {X 0,Y 403.57,Z 616.64,A -85,B 0,C 180,E1 -10893.993,E2 -10893.993} C_VEL
LIN {X 0,Y 403.441,Z 613.009,A -85,B 0,C 180,E1 -10895.998,E2 -10895.998} C_VEL
LIN {X 0,Y 403.422,Z 609.208,A -85,B 0,C 180,E1 -10897.506,E2 -10897.506} C_VEL
LIN {X 0,Y 403.432,Z 604.437,A -85,B 0,C 180,E1 -10899.019,E2 -10899.019} C_VEL
LIN {X 0,Y 403.674,Z 597.475,A -85,B 0,C 180,E1 -10900.786,E2 -10900.786} C_VEL
LIN {X 0,Y 404.011,Z 588.797,A -85,B 0,C 180,E1 -10902.558,E2 -10902.558} C_VEL
LIN {X 0,Y 404.635,Z 579.773,A -85,B 0,C 180,E1 -10904.072,E2 -10904.072} C_VEL
LIN {X 0,Y 405.495,Z 568.9,A -85,B 0,C 180,E1 -10905.582,E2 -10905.582} C_VEL
LIN {X 0,Y 406.384,Z 559.147,A -85,B 0,C 180,E1 -10906.708,E2 -10906.708} C_VEL
LIN {X 0,Y 407.293,Z 547.52,A -85,B 0,C 180,E1 -10907.834,E2 -10907.834} C_VEL
LIN {X 0,Y 408.266,Z 535.171,A -85,B 0,C 180,E1 -10908.812,E2 -10908.812} C_VEL
LIN {X 0,Y 408.783,Z 525.33,A -85,B 0,C 180,E1 -10909.456,E2 -10909.456} C_VEL
LIN {X 0,Y 407.383,Z 510.55,A -85,B 0,C 180,E1 -10910.296,E2 -10910.296} C_VEL
LIN {X 0,Y 405.453,Z 495.074,A -85,B 0,C 180,E1 -10910.974,E2 -10910.974} C_VEL
LIN {X 0,Y 404.133,Z 485.47,A -85,B 0,C 180,E1 -10911.299,E2 -10911.299} C_VEL
LIN {X 0,Y 404.721,Z 473.53,A -85,B 0,C 180,E1 -10914.629,E2 -10914.629} C_VEL
LIN {X 0,Y 405.386,Z 461.966,A -85,B 0,C 180,E1 -10917.909,E2 -10917.909} C_VEL
LIN {X 0,Y 406.306,Z 448.935,A -85,B 0,C 180,E1 -10921.669,E2 -10921.669} C_VEL
LIN {X 0,Y 407.131,Z 438.586,A -85,B 0,C 180,E1 -10924.724,E2 -10924.724} C_VEL
LIN {X 0,Y 408.362,Z 425.207,A -85,B 0,C 180,E1 -10928.784,E2 -10928.784} C_VEL
LIN {X 0,Y 408.529,Z 420.911,A -85,B 0,C 180,E1 -10930.129,E2 -10930.129} C_VEL
LIN {X 0,Y 407.466,Z 414.542,A -85,B 0,C 180,E1 -10932.272,E2 -10932.272} C_VEL
LIN {X 0,Y 405.188,Z 403.812,A -85,B 0,C 180,E1 -10936.068,E2 -10936.068} C_VEL
LIN {X 0,Y 404.198,Z 398.762,A -85,B 0,C 180,E1 -10937.967,E2 -10937.967} C_VEL
LIN {X 0,Y 404.155,Z 398.769,A -85,B 0,C 180,E1 -10941.49,E2 -10941.49} C_VEL
LIN {X 0,Y 404.177,Z 398.765,A -85,B 0,C 180,E1 -10944.983,E2 -10944.983} C_VEL
LIN {X 0,Y 404.136,Z 398.768,A -85,B 0,C 180,E1 -10948.553,E2 -10948.553} C_VEL
LIN {X 0,Y 404.188,Z 398.76,A -85,B 0,C 180,E1 -10952,E2 -10952} C_VEL
LIN {X 0,Y 404.167,Z 398.767,A -85,B 0,C 180,E1 -10955.334,E2 -10955.334} C_VEL
LIN {X 0,Y 404.128,Z 398.769,A -85,B 0,C 180,E1 -10958.58,E2 -10958.58} C_VEL
LIN {X 0,Y 404.2,Z 398.759,A -85,B 0,C 180,E1 -10961.762,E2 -10961.762} C_VEL
LIN {X 0,Y 404.197,Z 398.762,A -85,B 0,C 180,E1 -10964.882,E2 -10964.882} C_VEL
LIN {X 0,Y 404.26,Z 398.751,A -85,B 0,C 180,E1 -10967.959,E2 -10967.959} C_VEL
LIN {X 0,Y 404.422,Z 398.731,A -85,B 0,C 180,E1 -10972.1,E2 -10972.1} C_VEL
LIN {X 0,Y 404.413,Z 398.732,A -85,B 0,C 180,E1 -10974.015,E2 -10974.015} C_VEL
LIN {X 0,Y 404.473,Z 398.725,A -85,B 0,C 180,E1 -10978.009,E2 -10978.009} C_VEL
LIN {X 0,Y 404.603,Z 398.708,A -85,B 0,C 180,E1 -10980,E2 -10980} C_VEL
LIN {X 0,Y 404.415,Z 398.737,A -85,B 0,C 180,E1 -10982.989,E2 -10982.989} C_VEL
LIN {X 0,Y 404.402,Z 398.739,A -85,B 0,C 180,E1 -10986.988,E2 -10986.988} C_VEL
LIN {X 0,Y 404.262,Z 398.751,A -85,B 0,C 180,E1 -10990.012,E2 -10990.012} C_VEL
LIN {X 0,Y 404.256,Z 398.754,A -85,B 0,C 180,E1 -10993.212,E2 -10993.212} C_VEL
LIN {X 0,Y 404.206,Z 398.762,A -85,B 0,C 180,E1 -10997.008,E2 -10997.008} C_VEL
LIN {X 0,Y 404.154,Z 398.767,A -85,B 0,C 180,E1 -11000.352,E2 -11000.352} C_VEL
LIN {X 0,Y 404.16,Z 398.764,A -85,B 0,C 180,E1 -11003.575,E2 -11003.575} C_VEL
LIN {X 0,Y 404.175,Z 398.762,A -85,B 0,C 180,E1 -11005.767,E2 -11005.767} C_VEL
LIN {X 0,Y 404.187,Z 398.761,A -85,B 0,C 180,E1 -11008.001,E2 -11008.001} C_VEL
LIN {X 0,Y 404.131,Z 398.767,A -85,B 0,C 180,E1 -11011.559,E2 -11011.559} C_VEL
LIN {X 0,Y 404.178,Z 398.764,A -85,B 0,C 180,E1 -11015.017,E2 -11015.017} C_VEL
LIN {X 0,Y 404.153,Z 398.769,A -85,B 0,C 180,E1 -11018.758,E2 -11018.758} C_VEL
LIN {X 0,Y 404.119,Z 398.769,A -85,B 0,C 180,E1 -11021.601,E2 -11021.601} C_VEL
LIN {X 0,Y 404.144,Z 398.77,A -85,B 0,C 180,E1 -11024.524,E2 -11024.524} C_VEL
LIN {X 0,Y 404.166,Z 398.763,A -85,B 0,C 180,E1 -11027.302,E2 -11027.302} C_VEL
LIN {X 0,Y 404.165,Z 398.765,A -85,B 0,C 180,E1 -11029.957,E2 -11029.957} C_VEL
LIN {X 0,Y 404.138,Z 398.767,A -85,B 0,C 180,E1 -11033.126,E2 -11033.126} C_VEL
LIN {X 0,Y 404.143,Z 398.769,A -85,B 0,C 180,E1 -11036.189,E2 -11036.189} C_VEL
LIN {X 0,Y 404.144,Z 398.766,A -85,B 0,C 180,E1 -11039.716,E2 -11039.716} C_VEL
LIN {X 0,Y 404.195,Z 398.76,A -85,B 0,C 180,E1 -11043.124,E2 -11043.124} C_VEL
LIN {X 0,Y 404.177,Z 398.761,A -85,B 0,C 180,E1 -11045.336,E2 -11045.336} C_VEL
LIN {X 0,Y 404.14,Z 398.77,A -85,B 0,C 180,E1 -11048.582,E2 -11048.582} C_VEL
LIN {X 0,Y 404.209,Z 398.759,A -85,B 0,C 180,E1 -11051.763,E2 -11051.763} C_VEL
LIN {X 0,Y 404.122,Z 398.771,A -85,B 0,C 180,E1 -11054.88,E2 -11054.88} C_VEL
LIN {X 0,Y 404.132,Z 398.77,A -85,B 0,C 180,E1 -11055.435,E2 -11055.435} C_VEL
LIN {X 0,Y 408.23,Z 411.536,A -85,B 0,C 180,E1 -11056.026,E2 -11056.026} C_VEL
LIN {X 0,Y 409.418,Z 415.977,A -85,B 0,C 180,E1 -11056.273,E2 -11056.273} C_VEL
LIN {X 0,Y 409.029,Z 428.301,A -85,B 0,C 180,E1 -11056.93,E2 -11056.93} C_VEL
LIN {X 0,Y 408.5,Z 440.757,A -85,B 0,C 180,E1 -11057.835,E2 -11057.835} C_VEL
LIN {X 0,Y 407.888,Z 451.428,A -85,B 0,C 180,E1 -11058.824,E2 -11058.824} C_VEL
LIN {X 0,Y 407.217,Z 460.874,A -85,B 0,C 180,E1 -11059.908,E2 -11059.908} C_VEL
LIN {X 0,Y 406.434,Z 470.612,A -85,B 0,C 180,E1 -11061.299,E2 -11061.299} C_VEL
LIN {X 0,Y 405.856,Z 478.965,A -85,B 0,C 180,E1 -11062.789,E2 -11062.789} C_VEL
LIN {X 0,Y 405.272,Z 484.648,A -85,B 0,C 180,E1 -11064.029,E2 -11064.029} C_VEL
LIN {X 0,Y 404.954,Z 490.192,A -85,B 0,C 180,E1 -11065.522,E2 -11065.522} C_VEL
LIN {X 0,Y 404.579,Z 494.558,A -85,B 0,C 180,E1 -11067.014,E2 -11067.014} C_VEL
LIN {X 0,Y 404.38,Z 496.852,A -85,B 0,C 180,E1 -11068.009,E2 -11068.009} C_VEL
LIN {X 0,Y 404.125,Z 500.209,A -85,B 0,C 180,E1 -11070.001,E2 -11070.001} C_VEL
LIN {X 0,Y 403.958,Z 501.268,A -85,B 0,C 180,E1 -11070.998,E2 -11070.998} C_VEL
LIN {X 0,Y 404.024,Z 501.91,A -85,B 0,C 180,E1 -11071.995,E2 -11071.995} C_VEL
LIN {X 0,Y 403.89,Z 502.217,A -85,B 0,C 180,E1 -11072.993,E2 -11072.993} C_VEL
LIN {X 0,Y 403.958,Z 502.122,A -85,B 0,C 180,E1 -11073.992,E2 -11073.992} C_VEL
LIN {X 0,Y 404.302,Z 500.692,A -85,B 0,C 180,E1 -11075.988,E2 -11075.988} C_VEL
LIN {X 0,Y 404.37,Z 499.429,A -85,B 0,C 180,E1 -11076.989,E2 -11076.989} C_VEL
LIN {X 0,Y 404.664,Z 496.383,A -85,B 0,C 180,E1 -11078.637,E2 -11078.637} C_VEL
LIN {X 0,Y 405.093,Z 492.979,A -85,B 0,C 180,E1 -11079.992,E2 -11079.992} C_VEL
LIN {X 0,Y 405.554,Z 488.142,A -85,B 0,C 180,E1 -11081.496,E2 -11081.496} C_VEL
LIN {X 0,Y 405.904,Z 483.853,A -85,B 0,C 180,E1 -11082.581,E2 -11082.581} C_VEL
LIN {X 0,Y 405.504,Z 480.839,A -85,B 0,C 180,E1 -11083.297,E2 -11083.297} C_VEL
LIN {X 0,Y 403.22,Z 475.724,A -85,B 0,C 180,E1 -11084.458,E2 -11084.458} C_VEL
LIN {X 0,Y 401.01,Z 470.079,A -85,B 0,C 180,E1 -11085.57,E2 -11085.57} C_VEL
LIN {X 0,Y 400.718,Z 466.1,A -85,B 0,C 180,E1 -11086.197,E2 -11086.197} C_VEL
LIN {X 0,Y 401.515,Z 456.354,A -85,B 0,C 180,E1 -11087.444,E2 -11087.444} C_VEL
LIN {X 0,Y 402.26,Z 445.12,A -85,B 0,C 180,E1 -11088.594,E2 -11088.594} C_VEL
LIN {X 0,Y 402.875,Z 433.69,A -85,B 0,C 180,E1 -11089.508,E2 -11089.508} C_VEL
LIN {X 0,Y 403.377,Z 421.589,A -85,B 0,C 180,E1 -11090.243,E2 -11090.243} C_VEL
LIN {X 0,Y 403.287,Z 417.626,A -85,B 0,C 180,E1 -11090.45,E2 -11090.45} C_VEL
LIN {X 0,Y 399.229,Z 405.864,A -85,B 0,C 180,E1 -11091.141,E2 -11091.141} C_VEL
LIN {X 0,Y 397.028,Z 399.656,A -85,B 0,C 180,E1 -11091.447,E2 -11091.447} C_VEL
LIN {X 0,Y 397.134,Z 399.64,A -85,B 0,C 180,E1 -11094.019,E2 -11094.019} C_VEL
LIN {X 0,Y 397.2,Z 399.634,A -85,B 0,C 180,E1 -11097.391,E2 -11097.391} C_VEL
LIN {X 0,Y 397.085,Z 399.65,A -85,B 0,C 180,E1 -11100.883,E2 -11100.883} C_VEL
LIN {X 0,Y 397.13,Z 399.645,A -85,B 0,C 180,E1 -11104.494,E2 -11104.494} C_VEL
LIN {X 0,Y 397.107,Z 399.634,A -85,B 0,C 180,E1 -11108.275,E2 -11108.275} C_VEL
LIN {X 0,Y 397.094,Z 399.647,A -85,B 0,C 180,E1 -11110.909,E2 -11110.909} C_VEL
LIN {X 0,Y 397.107,Z 399.642,A -85,B 0,C 180,E1 -11113.649,E2 -11113.649} C_VEL
LIN {X 0,Y 397.112,Z 399.645,A -85,B 0,C 180,E1 -11116.52,E2 -11116.52} C_VEL
LIN {X 0,Y 397.119,Z 399.621,A -85,B 0,C 180,E1 -11120.423,E2 -11120.423} C_VEL
LIN {X 0,Y 397.114,Z 399.644,A -85,B 0,C 180,E1 -11124.266,E2 -11124.266} C_VEL
LIN {X 0,Y 397.119,Z 399.638,A -85,B 0,C 180,E1 -11126.727,E2 -11126.727} C_VEL
LIN {X 0,Y 397.129,Z 399.609,A -85,B 0,C 180,E1 -11130.296,E2 -11130.296} C_VEL
LIN {X 0,Y 397.199,Z 399.621,A -85,B 0,C 180,E1 -11132.61,E2 -11132.61} C_VEL
LIN {X 0,Y 397.133,Z 399.643,A -85,B 0,C 180,E1 -11135.981,E2 -11135.981} C_VEL
LIN {X 0,Y 397.143,Z 399.642,A -85,B 0,C 180,E1 -11139.705,E2 -11139.705} C_VEL
LIN {X 0,Y 397.139,Z 399.64,A -85,B 0,C 180,E1 -11140.806,E2 -11140.806} C_VEL
LIN {X 0,Y 401.211,Z 413.196,A -85,B 0,C 180,E1 -11141.839,E2 -11141.839} C_VEL
LIN {X 0,Y 402.921,Z 419.405,A -85,B 0,C 180,E1 -11142.375,E2 -11142.375} C_VEL
LIN {X 0,Y 402.082,Z 432.788,A -85,B 0,C 180,E1 -11143.499,E2 -11143.499} C_VEL
LIN {X 0,Y 401.204,Z 445.006,A -85,B 0,C 180,E1 -11144.766,E2 -11144.766} C_VEL
LIN {X 0,Y 400.348,Z 455.171,A -85,B 0,C 180,E1 -11146.032,E2 -11146.032} C_VEL
LIN {X 0,Y 399.491,Z 465.339,A -85,B 0,C 180,E1 -11147.554,E2 -11147.554} C_VEL
LIN {X 0,Y 398.771,Z 475.086,A -85,B 0,C 180,E1 -11149.335,E2 -11149.335} C_VEL
LIN {X 0,Y 398.158,Z 483.025,A -85,B 0,C 180,E1 -11151.115,E2 -11151.115} C_VEL
LIN {X 0,Y 397.696,Z 489.428,A -85,B 0,C 180,E1 -11152.894,E2 -11152.894} C_VEL
LIN {X 0,Y 397.473,Z 493.8,A -85,B 0,C 180,E1 -11154.419,E2 -11154.419} C_VEL
LIN {X 0,Y 397.077,Z 497.342,A -85,B 0,C 180,E1 -11155.94,E2 -11155.94} C_VEL
LIN {X 0,Y 397.016,Z 500.719,A -85,B 0,C 180,E1 -11157.971,E2 -11157.971} C_VEL
LIN {X 0,Y 397.022,Z 502.726,A -85,B 0,C 180,E1 -11160,E2 -11160} C_VEL
LIN {X 0,Y 397.167,Z 503.381,A -85,B 0,C 180,E1 -11162.028,E2 -11162.028} C_VEL
LIN {X 0,Y 397.288,Z 502.732,A -85,B 0,C 180,E1 -11164.057,E2 -11164.057} C_VEL
LIN {X 0,Y 397.621,Z 500.723,A -85,B 0,C 180,E1 -11166.087,E2 -11166.087} C_VEL
LIN {X 0,Y 398.208,Z 497.249,A -85,B 0,C 180,E1 -11168.117,E2 -11168.117} C_VEL
LIN {X 0,Y 398.892,Z 492.266,A -85,B 0,C 180,E1 -11170.148,E2 -11170.148} C_VEL
LIN {X 0,Y 399.761,Z 485.649,A -85,B 0,C 180,E1 -11172.179,E2 -11172.179} C_VEL
LIN {X 0,Y 400.771,Z 478.248,A -85,B 0,C 180,E1 -11173.953,E2 -11173.953} C_VEL
LIN {X 0,Y 401.851,Z 470.587,A -85,B 0,C 180,E1 -11175.443,E2 -11175.443} C_VEL
LIN {X 0,Y 403.049,Z 460.997,A -85,B 0,C 180,E1 -11176.982,E2 -11176.982} C_VEL
LIN {X 0,Y 404.189,Z 450.635,A -85,B 0,C 180,E1 -11178.37,E2 -11178.37} C_VEL
LIN {X 0,Y 405.368,Z 439.219,A -85,B 0,C 180,E1 -11179.628,E2 -11179.628} C_VEL
LIN {X 0,Y 406.481,Z 427.406,A -85,B 0,C 180,E1 -11180.688,E2 -11180.688} C_VEL
LIN {X 0,Y 406.578,Z 423.349,A -85,B 0,C 180,E1 -11181.023,E2 -11181.023} C_VEL
LIN {X 0,Y 402.915,Z 412.929,A -85,B 0,C 180,E1 -11182.146,E2 -11182.146} C_VEL
LIN {X 0,Y 398.686,Z 403.267,A -85,B 0,C 180,E1 -11183.172,E2 -11183.172} C_VEL
LIN {X 0,Y 397.402,Z 400.905,A -85,B 0,C 180,E1 -11183.436,E2 -11183.436} C_VEL
LIN {X 0,Y 397.136,Z 399.645,A -85,B 0,C 180,E1 -11183.538,E2 -11183.538} C_VEL
LIN {X 0,Y 397.139,Z 399.644,A -85,B 0,C 180,E1 -11186.258,E2 -11186.258} C_VEL
LIN {X 0,Y 397.125,Z 399.641,A -85,B 0,C 180,E1 -11188.543,E2 -11188.543} C_VEL
LIN {X 0,Y 397.081,Z 399.647,A -85,B 0,C 180,E1 -11192.071,E2 -11192.071} C_VEL
LIN {X 0,Y 397.122,Z 399.644,A -85,B 0,C 180,E1 -11195.503,E2 -11195.503} C_VEL
LIN {X 0,Y 397.133,Z 399.643,A -85,B 0,C 180,E1 -11198.861,E2 -11198.861} C_VEL
LIN {X 0,Y 397.111,Z 399.778,A -85,B 0,C 180,E1 -11201.464,E2 -11201.464} C_VEL
LIN {X 0,Y 398.041,Z 404.015,A -85,B 0,C 180,E1 -11204.22,E2 -11204.22} C_VEL
LIN {X 0,Y 399.149,Z 409.338,A -85,B 0,C 180,E1 -11207.049,E2 -11207.049} C_VEL
LIN {X 0,Y 400.162,Z 414.71,A -85,B 0,C 180,E1 -11209.471,E2 -11209.471} C_VEL
LIN {X 0,Y 400.374,Z 418.078,A -85,B 0,C 180,E1 -11210.807,E2 -11210.807} C_VEL
LIN {X 0,Y 398.911,Z 428.771,A -85,B 0,C 180,E1 -11214.451,E2 -11214.451} C_VEL
LIN {X 0,Y 398.271,Z 438.256,A -85,B 0,C 180,E1 -11217.433,E2 -11217.433} C_VEL
LIN {X 0,Y 397.815,Z 448.126,A -85,B 0,C 180,E1 -11220.352,E2 -11220.352} C_VEL
LIN {X 0,Y 397.265,Z 461.712,A -85,B 0,C 180,E1 -11224.161,E2 -11224.161} C_VEL
LIN {X 0,Y 396.973,Z 471.443,A -85,B 0,C 180,E1 -11226.794,E2 -11226.794} C_VEL
LIN {X 0,Y 400.161,Z 488.923,A -85,B 0,C 180,E1 -11227.721,E2 -11227.721} C_VEL
LIN {X 0,Y 401.534,Z 502.524,A -85,B 0,C 180,E1 -11228.497,E2 -11228.497} C_VEL
LIN {X 0,Y 401.85,Z 517.211,A -85,B 0,C 180,E1 -11229.426,E2 -11229.426} C_VEL
LIN {X 0,Y 402.195,Z 529.227,A -85,B 0,C 180,E1 -11230.343,E2 -11230.343} C_VEL
LIN {X 0,Y 400.887,Z 542.151,A -85,B 0,C 180,E1 -11231.421,E2 -11231.421} C_VEL
LIN {X 0,Y 399.689,Z 553.979,A -85,B 0,C 180,E1 -11232.606,E2 -11232.606} C_VEL
LIN {X 0,Y 398.454,Z 566.61,A -85,B 0,C 180,E1 -11234.133,E2 -11234.133} C_VEL
LIN {X 0,Y 397.609,Z 577.227,A -85,B 0,C 180,E1 -11235.672,E2 -11235.672} C_VEL
LIN {X 0,Y 396.929,Z 587.672,A -85,B 0,C 180,E1 -11237.493,E2 -11237.493} C_VEL
LIN {X 0,Y 396.585,Z 596.074,A -85,B 0,C 180,E1 -11239.275,E2 -11239.275} C_VEL
LIN {X 0,Y 396.433,Z 602.074,A -85,B 0,C 180,E1 -11240.818,E2 -11240.818} C_VEL
LIN {X 0,Y 396.416,Z 608.514,A -85,B 0,C 180,E1 -11242.87,E2 -11242.87} C_VEL
LIN {X 0,Y 396.59,Z 613.265,A -85,B 0,C 180,E1 -11244.916,E2 -11244.916} C_VEL
LIN {X 0,Y 396.614,Z 615.019,A -85,B 0,C 180,E1 -11245.934,E2 -11245.934} C_VEL
LIN {X 0,Y 396.606,Z 617.378,A -85,B 0,C 180,E1 -11247.968,E2 -11247.968} C_VEL
LIN {X 0,Y 396.744,Z 618.021,A -85,B 0,C 180,E1 -11248.984,E2 -11248.984} C_VEL
LIN {X 0,Y 396.825,Z 618.284,A -85,B 0,C 180,E1 -11249.999,E2 -11249.999} C_VEL
LIN {X 0,Y 396.575,Z 617.632,A -85,B 0,C 180,E1 -11252.03,E2 -11252.03} C_VEL
LIN {X 0,Y 396.535,Z 615.523,A -85,B 0,C 180,E1 -11254.064,E2 -11254.064} C_VEL
LIN {X 0,Y 396.429,Z 612.923,A -85,B 0,C 180,E1 -11255.594,E2 -11255.594} C_VEL
LIN {X 0,Y 396.362,Z 608.009,A -85,B 0,C 180,E1 -11257.641,E2 -11257.641} C_VEL
LIN {X 0,Y 396.392,Z 603.189,A -85,B 0,C 180,E1 -11259.181,E2 -11259.181} C_VEL
LIN {X 0,Y 396.627,Z 596.165,A -85,B 0,C 180,E1 -11260.98,E2 -11260.98} C_VEL
LIN {X 0,Y 396.966,Z 587.619,A -85,B 0,C 180,E1 -11262.747,E2 -11262.747} C_VEL
LIN {X 0,Y 397.67,Z 578.33,A -85,B 0,C 180,E1 -11264.324,E2 -11264.324} C_VEL
LIN {X 0,Y 398.543,Z 567.371,A -85,B 0,C 180,E1 -11265.861,E2 -11265.861} C_VEL
LIN {X 0,Y 399.549,Z 556.347,A -85,B 0,C 180,E1 -11267.134,E2 -11267.134} C_VEL
LIN {X 0,Y 400.613,Z 544.35,A -85,B 0,C 180,E1 -11268.274,E2 -11268.274} C_VEL
LIN {X 0,Y 401.548,Z 531.842,A -85,B 0,C 180,E1 -11269.243,E2 -11269.243} C_VEL
LIN {X 0,Y 401.855,Z 526.42,A -85,B 0,C 180,E1 -11269.606,E2 -11269.606} C_VEL
LIN {X 0,Y 400.537,Z 511.936,A -85,B 0,C 180,E1 -11270.476,E2 -11270.476} C_VEL
LIN {X 0,Y 398.721,Z 496.737,A -85,B 0,C 180,E1 -11271.183,E2 -11271.183} C_VEL
LIN {X 0,Y 397.127,Z 484.663,A -85,B 0,C 180,E1 -11271.612,E2 -11271.612} C_VEL
LIN {X 0,Y 397.733,Z 472.466,A -85,B 0,C 180,E1 -11275.091,E2 -11275.091} C_VEL
LIN {X 0,Y 398.431,Z 460.915,A -85,B 0,C 180,E1 -11278.44,E2 -11278.44} C_VEL
LIN {X 0,Y 399.297,Z 449.285,A -85,B 0,C 180,E1 -11281.871,E2 -11281.871} C_VEL
LIN {X 0,Y 400.132,Z 439.483,A -85,B 0,C 180,E1 -11284.819,E2 -11284.819} C_VEL
LIN {X 0,Y 401.258,Z 427.69,A -85,B 0,C 180,E1 -11288.453,E2 -11288.453} C_VEL
LIN {X 0,Y 401.607,Z 422.973,A -85,B 0,C 180,E1 -11289.945,E2 -11289.945} C_VEL
LIN {X 0,Y 400.61,Z 416.494,A -85,B 0,C 180,E1 -11292.143,E2 -11292.143} C_VEL
LIN {X 0,Y 398.461,Z 406.167,A -85,B 0,C 180,E1 -11295.838,E2 -11295.838} C_VEL
LIN {X 0,Y 397.157,Z 399.639,A -85,B 0,C 180,E1 -11298.321,E2 -11298.321} C_VEL
LIN {X 0,Y 397.102,Z 399.647,A -85,B 0,C 180,E1 -11301.725,E2 -11301.725} C_VEL
LIN {X 0,Y 397.117,Z 399.644,A -85,B 0,C 180,E1 -11305.506,E2 -11305.506} C_VEL
LIN {X 0,Y 397.076,Z 399.65,A -85,B 0,C 180,E1 -11309.117,E2 -11309.117} C_VEL
LIN {X 0,Y 397.185,Z 399.634,A -85,B 0,C 180,E1 -11312.609,E2 -11312.609} C_VEL
LIN {X 0,Y 397.123,Z 399.64,A -85,B 0,C 180,E1 -11315.981,E2 -11315.981} C_VEL
LIN {X 0,Y 397.128,Z 399.64,A -85,B 0,C 180,E1 -11319.704,E2 -11319.704} C_VEL
LIN {X 0,Y 397.171,Z 399.638,A -85,B 0,C 180,E1 -11322.845,E2 -11322.845} C_VEL
LIN {X 0,Y 397.215,Z 399.632,A -85,B 0,C 180,E1 -11326.679,E2 -11326.679} C_VEL
LIN {X 0,Y 397.219,Z 399.628,A -85,B 0,C 180,E1 -11329.809,E2 -11329.809} C_VEL
LIN {X 0,Y 397.353,Z 399.616,A -85,B 0,C 180,E1 -11332.888,E2 -11332.888} C_VEL
LIN {X 0,Y 397.247,Z 399.629,A -85,B 0,C 180,E1 -11334.925,E2 -11334.925} C_VEL
LIN {X 0,Y 397.442,Z 399.6,A -85,B 0,C 180,E1 -11337.973,E2 -11337.973} C_VEL
LIN {X 0,Y 397.572,Z 399.584,A -85,B 0,C 180,E1 -11340,E2 -11340} C_VEL
LIN {X 0,Y 397.373,Z 399.614,A -85,B 0,C 180,E1 -11343.042,E2 -11343.042} C_VEL
LIN {X 0,Y 397.354,Z 399.615,A -85,B 0,C 180,E1 -11347.112,E2 -11347.112} C_VEL
LIN {X 0,Y 397.22,Z 399.629,A -85,B 0,C 180,E1 -11350.191,E2 -11350.191} C_VEL
LIN {X 0,Y 397.216,Z 399.63,A -85,B 0,C 180,E1 -11353.322,E2 -11353.322} C_VEL
LIN {X 0,Y 397.172,Z 399.636,A -85,B 0,C 180,E1 -11357.156,E2 -11357.156} C_VEL
LIN {X 0,Y 397.093,Z 399.648,A -85,B 0,C 180,E1 -11360.731,E2 -11360.731} C_VEL
LIN {X 0,Y 397.124,Z 399.641,A -85,B 0,C 180,E1 -11364.019,E2 -11364.019} C_VEL
LIN {X 0,Y 397.186,Z 399.633,A -85,B 0,C 180,E1 -11367.391,E2 -11367.391} C_VEL
LIN {X 0,Y 397.071,Z 399.651,A -85,B 0,C 180,E1 -11370.884,E2 -11370.884} C_VEL
LIN {X 0,Y 397.119,Z 399.645,A -85,B 0,C 180,E1 -11374.494,E2 -11374.494} C_VEL
LIN {X 0,Y 397.1,Z 399.646,A -85,B 0,C 180,E1 -11378.276,E2 -11378.276} C_VEL
LIN {X 0,Y 397.084,Z 399.648,A -85,B 0,C 180,E1 -11380.91,E2 -11380.91} C_VEL
LIN {X 0,Y 397.099,Z 399.643,A -85,B 0,C 180,E1 -11383.649,E2 -11383.649} C_VEL
LIN {X 0,Y 397.1,Z 399.648,A -85,B 0,C 180,E1 -11386.522,E2 -11386.522} C_VEL
LIN {X 0,Y 397.117,Z 399.641,A -85,B 0,C 180,E1 -11389.553,E2 -11389.553} C_VEL
LIN {X 0,Y 397.096,Z 399.647,A -85,B 0,C 180,E1 -11392.791,E2 -11392.791} C_VEL
LIN {X 0,Y 397.116,Z 399.645,A -85,B 0,C 180,E1 -11396.284,E2 -11396.284} C_VEL
LIN {X 0,Y 397.104,Z 399.646,A -85,B 0,C 180,E1 -11400.137,E2 -11400.137} C_VEL
LIN {X 0,Y 397.194,Z 399.635,A -85,B 0,C 180,E1 -11402.611,E2 -11402.611} C_VEL
LIN {X 0,Y 397.133,Z 399.642,A -85,B 0,C 180,E1 -11405.983,E2 -11405.983} C_VEL
LIN {X 0,Y 397.139,Z 399.639,A -85,B 0,C 180,E1 -11409.706,E2 -11409.706} C_VEL
LIN {X 0,Y 397.177,Z 399.635,A -85,B 0,C 180,E1 -11412.849,E2 -11412.849} C_VEL
LIN {X 0,Y 397.082,Z 399.647,A -85,B 0,C 180,E1 -11415.132,E2 -11415.132} C_VEL
LIN {X 0,Y 401.155,Z 412.051,A -85,B 0,C 180,E1 -11415.719,E2 -11415.719} C_VEL
LIN {X 0,Y 402.626,Z 417.7,A -85,B 0,C 180,E1 -11416.037,E2 -11416.037} C_VEL
LIN {X 0,Y 402.205,Z 429.81,A -85,B 0,C 180,E1 -11416.704,E2 -11416.704} C_VEL
LIN {X 0,Y 401.686,Z 442.141,A -85,B 0,C 180,E1 -11417.625,E2 -11417.625} C_VEL
LIN {X 0,Y 401.036,Z 452.747,A -85,B 0,C 180,E1 -11418.631,E2 -11418.631} C_VEL
LIN {X 0,Y 400.394,Z 461.343,A -85,B 0,C 180,E1 -11419.632,E2 -11419.632} C_VEL
LIN {X 0,Y 399.689,Z 470.255,A -85,B 0,C 180,E1 -11420.896,E2 -11420.896} C_VEL
LIN {X 0,Y 399.044,Z 478.839,A -85,B 0,C 180,E1 -11422.411,E2 -11422.411} C_VEL
LIN {X 0,Y 398.303,Z 485.792,A -85,B 0,C 180,E1 -11423.924,E2 -11423.924} C_VEL
LIN {X 0,Y 397.962,Z 491.304,A -85,B 0,C 180,E1 -11425.443,E2 -11425.443} C_VEL
LIN {X 0,Y 397.576,Z 495.643,A -85,B 0,C 180,E1 -11426.961,E2 -11426.961} C_VEL
LIN {X 0,Y 397.367,Z 497.923,A -85,B 0,C 180,E1 -11427.974,E2 -11427.974} C_VEL
LIN {X 0,Y 397.105,Z 501.255,A -85,B 0,C 180,E1 -11430.001,E2 -11430.001} C_VEL
LIN {X 0,Y 396.934,Z 502.297,A -85,B 0,C 180,E1 -11431.016,E2 -11431.016} C_VEL
LIN {X 0,Y 397.001,Z 502.929,A -85,B 0,C 180,E1 -11432.03,E2 -11432.03} C_VEL
LIN {X 0,Y 396.865,Z 503.227,A -85,B 0,C 180,E1 -11433.046,E2 -11433.046} C_VEL
LIN {X 0,Y 396.937,Z 503.115,A -85,B 0,C 180,E1 -11434.062,E2 -11434.062} C_VEL
LIN {X 0,Y 397.306,Z 501.659,A -85,B 0,C 180,E1 -11436.094,E2 -11436.094} C_VEL
LIN {X 0,Y 397.384,Z 500.386,A -85,B 0,C 180,E1 -11437.112,E2 -11437.112} C_VEL
LIN {X 0,Y 397.661,Z 497.651,A -85,B 0,C 180,E1 -11438.641,E2 -11438.641} C_VEL
LIN {X 0,Y 398.138,Z 493.893,A -85,B 0,C 180,E1 -11440.168,E2 -11440.168} C_VEL
LIN {X 0,Y 398.644,Z 489.026,A -85,B 0,C 180,E1 -11441.698,E2 -11441.698} C_VEL
LIN {X 0,Y 399.182,Z 482.856,A -85,B 0,C 180,E1 -11443.232,E2 -11443.232} C_VEL
LIN {X 0,Y 399.759,Z 476.297,A -85,B 0,C 180,E1 -11444.556,E2 -11444.556} C_VEL
LIN {X 0,Y 400.63,Z 467.19,A -85,B 0,C 180,E1 -11446.04,E2 -11446.04} C_VEL
LIN {X 0,Y 400.718,Z 466.1,A -85,B 0,C 180,E1 -11446.197,E2 -11446.197} C_VEL
LIN {X 0,Y 400.425,Z 461.968,A -85,B 0,C 180,E1 -11446.802,E2 -11446.802} C_VEL
LIN {X 0,Y 398.232,Z 455.127,A -85,B 0,C 180,E1 -11447.786,E2 -11447.786} C_VEL
LIN {X 0,Y 396.032,Z 447.81,A -85,B 0,C 180,E1 -11448.693,E2 -11448.693} C_VEL
LIN {X 0,Y 395.713,Z 442.921,A -85,B 0,C 180,E1 -11449.169,E2 -11449.169} C_VEL
LIN {X 0,Y 396.312,Z 432.445,A -85,B 0,C 180,E1 -11449.968,E2 -11449.968} C_VEL
LIN {X 0,Y 396.808,Z 420.176,A -85,B 0,C 180,E1 -11450.687,E2 -11450.687} C_VEL
LIN {X 0,Y 392.942,Z 408.606,A -85,B 0,C 180,E1 -11451.4,E2 -11451.4} C_VEL
LIN {X 0,Y 390.016,Z 400.528,A -85,B 0,C 180,E1 -11451.812,E2 -11451.812} C_VEL
LIN {X 0,Y 390.083,Z 400.518,A -85,B 0,C 180,E1 -11454.481,E2 -11454.481} C_VEL
LIN {X 0,Y 390.123,Z 400.513,A -85,B 0,C 180,E1 -11457.93,E2 -11457.93} C_VEL
LIN {X 0,Y 390.029,Z 400.528,A -85,B 0,C 180,E1 -11461.505,E2 -11461.505} C_VEL
LIN {X 0,Y 390.09,Z 400.521,A -85,B 0,C 180,E1 -11465.207,E2 -11465.207} C_VEL
LIN {X 0,Y 390.074,Z 400.516,A -85,B 0,C 180,E1 -11469.218,E2 -11469.218} C_VEL
LIN {X 0,Y 390.048,Z 400.523,A -85,B 0,C 180,E1 -11472.374,E2 -11472.374} C_VEL
LIN {X 0,Y 390.052,Z 400.518,A -85,B 0,C 180,E1 -11475.355,E2 -11475.355} C_VEL
LIN {X 0,Y 390.051,Z 400.524,A -85,B 0,C 180,E1 -11478.189,E2 -11478.189} C_VEL
LIN {X 0,Y 390.096,Z 400.492,A -85,B 0,C 180,E1 -11480.908,E2 -11480.908} C_VEL
LIN {X 0,Y 390.091,Z 400.517,A -85,B 0,C 180,E1 -11484.793,E2 -11484.793} C_VEL
LIN {X 0,Y 390.036,Z 400.514,A -85,B 0,C 180,E1 -11487.876,E2 -11487.876} C_VEL
LIN {X 0,Y 390.063,Z 400.49,A -85,B 0,C 180,E1 -11490.89,E2 -11490.89} C_VEL
LIN {X 0,Y 390.123,Z 400.513,A -85,B 0,C 180,E1 -11494.257,E2 -11494.257} C_VEL
LIN {X 0,Y 390.042,Z 400.527,A -85,B 0,C 180,E1 -11497.766,E2 -11497.766} C_VEL
LIN {X 0,Y 390.117,Z 400.514,A -85,B 0,C 180,E1 -11500.497,E2 -11500.497} C_VEL
LIN {X 0,Y 394.66,Z 415.713,A -85,B 0,C 180,E1 -11501.712,E2 -11501.712} C_VEL
LIN {X 0,Y 396.035,Z 421.112,A -85,B 0,C 180,E1 -11502.193,E2 -11502.193} C_VEL
LIN {X 0,Y 395.187,Z 434.334,A -85,B 0,C 180,E1 -11503.335,E2 -11503.335} C_VEL
LIN {X 0,Y 394.257,Z 446.42,A -85,B 0,C 180,E1 -11504.623,E2 -11504.623} C_VEL
LIN {X 0,Y 393.298,Z 457.424,A -85,B 0,C 180,E1 -11506.04,E2 -11506.04} C_VEL
LIN {X 0,Y 392.444,Z 467.407,A -85,B 0,C 180,E1 -11507.59,E2 -11507.59} C_VEL
LIN {X 0,Y 391.832,Z 475.726,A -85,B 0,C 180,E1 -11509.144,E2 -11509.144} C_VEL
LIN {X 0,Y 391.196,Z 483.799,A -85,B 0,C 180,E1 -11510.968,E2 -11510.968} C_VEL
LIN {X 0,Y 390.71,Z 490.226,A -85,B 0,C 180,E1 -11512.766,E2 -11512.766} C_VEL
LIN {X 0,Y 390.481,Z 494.669,A -85,B 0,C 180,E1 -11514.319,E2 -11514.319} C_VEL
LIN {X 0,Y 390.057,Z 498.271,A -85,B 0,C 180,E1 -11515.867,E2 -11515.867} C_VEL
LIN {X 0,Y 389.994,Z 501.709,A -85,B 0,C 180,E1 -11517.934,E2 -11517.934} C_VEL
LIN {X 0,Y 390.01,Z 503.776,A -85,B 0,C 180,E1 -11520,E2 -11520} C_VEL
LIN {X 0,Y 390.164,Z 504.501,A -85,B 0,C 180,E1 -11522.064,E2 -11522.064} C_VEL
LIN {X 0,Y 390.311,Z 503.915,A -85,B 0,C 180,E1 -11524.13,E2 -11524.13} C_VEL
LIN {X 0,Y 390.669,Z 501.97,A -85,B 0,C 180,E1 -11526.196,E2 -11526.196} C_VEL
LIN {X 0,Y 391.297,Z 498.563,A -85,B 0,C 180,E1 -11528.261,E2 -11528.261} C_VEL
LIN {X 0,Y 392.064,Z 493.677,A -85,B 0,C 180,E1 -11530.326,E2 -11530.326} C_VEL
LIN {X 0,Y 392.725,Z 488.962,A -85,B 0,C 180,E1 -11531.876,E2 -11531.876} C_VEL
LIN {X 0,Y 393.74,Z 482.064,A -85,B 0,C 180,E1 -11533.68,E2 -11533.68} C_VEL
LIN {X 0,Y 395.01,Z 473.484,A -85,B 0,C 180,E1 -11535.478,E2 -11535.478} C_VEL
LIN {X 0,Y 396.275,Z 464.556,A -85,B 0,C 180,E1 -11537.015,E2 -11537.015} C_VEL
LIN {X 0,Y 397.346,Z 455.664,A -85,B 0,C 180,E1 -11538.297,E2 -11538.297} C_VEL
LIN {X 0,Y 398.707,Z 443.901,A -85,B 0,C 180,E1 -11539.701,E2 -11539.701} C_VEL
LIN {X 0,Y 399.961,Z 431.56,A -85,B 0,C 180,E1 -11540.895,E2 -11540.895} C_VEL
LIN {X 0,Y 400.433,Z 426.091,A -85,B 0,C 180,E1 -11541.352,E2 -11541.352} C_VEL
LIN {X 0,Y 397.034,Z 416.219,A -85,B 0,C 180,E1 -11542.483,E2 -11542.483} C_VEL
LIN {X 0,Y 392.93,Z 406.869,A -85,B 0,C 180,E1 -11543.555,E2 -11543.555} C_VEL
LIN {X 0,Y 390.575,Z 402.291,A -85,B 0,C 180,E1 -11544.086,E2 -11544.086} C_VEL
LIN {X 0,Y 390.093,Z 400.525,A -85,B 0,C 180,E1 -11544.271,E2 -11544.271} C_VEL
LIN {X 0,Y 390.117,Z 400.519,A -85,B 0,C 180,E1 -11546.768,E2 -11546.768} C_VEL
LIN {X 0,Y 390.042,Z 400.524,A -85,B 0,C 180,E1 -11550.299,E2 -11550.299} C_VEL
LIN {X 0,Y 390.071,Z 400.522,A -85,B 0,C 180,E1 -11554.024,E2 -11554.024} C_VEL
LIN {X 0,Y 390.046,Z 400.525,A -85,B 0,C 180,E1 -11557.55,E2 -11557.55} C_VEL
LIN {X 0,Y 390.068,Z 400.564,A -85,B 0,C 180,E1 -11560.438,E2 -11560.438} C_VEL
LIN {X 0,Y 390.836,Z 404.293,A -85,B 0,C 180,E1 -11563.103,E2 -11563.103} C_VEL
LIN {X 0,Y 391.833,Z 408.973,A -85,B 0,C 180,E1 -11565.844,E2 -11565.844} C_VEL
LIN {X 0,Y 393.003,Z 414.79,A -85,B 0,C 180,E1 -11568.684,E2 -11568.684} C_VEL
LIN {X 0,Y 393.498,Z 418.265,A -85,B 0,C 180,E1 -11570.174,E2 -11570.174} C_VEL
LIN {X 0,Y 393.223,Z 421.184,A -85,B 0,C 180,E1 -11571.277,E2 -11571.277} C_VEL
LIN {X 0,Y 391.688,Z 433.916,A -85,B 0,C 180,E1 -11575.626,E2 -11575.626} C_VEL
LIN {X 0,Y 390.969,Z 445.317,A -85,B 0,C 180,E1 -11579.175,E2 -11579.175} C_VEL
LIN {X 0,Y 390.382,Z 457.269,A -85,B 0,C 180,E1 -11582.672,E2 -11582.672} C_VEL
LIN {X 0,Y 389.999,Z 469.536,A -85,B 0,C 180,E1 -11586.105,E2 -11586.105} C_VEL
LIN {X 0,Y 393.646,Z 488.959,A -85,B 0,C 180,E1 -11587.233,E2 -11587.233} C_VEL
LIN {X 0,Y 394.945,Z 502.513,A -85,B 0,C 180,E1 -11588.056,E2 -11588.056} C_VEL
LIN {X 0,Y 395.194,Z 517.457,A -85,B 0,C 180,E1 -11589.06,E2 -11589.06} C_VEL
LIN {X 0,Y 395.338,Z 530.722,A -85,B 0,C 180,E1 -11590.123,E2 -11590.123} C_VEL
LIN {X 0,Y 393.759,Z 544.88,A -85,B 0,C 180,E1 -11591.394,E2 -11591.394} C_VEL
LIN {X 0,Y 392.406,Z 557.846,A -85,B 0,C 180,E1 -11592.811,E2 -11592.811} C_VEL
LIN {X 0,Y 391.214,Z 569.608,A -85,B 0,C 180,E1 -11594.366,E2 -11594.366} C_VEL
LIN {X 0,Y 390.433,Z 579.543,A -85,B 0,C 180,E1 -11595.935,E2 -11595.935} C_VEL
LIN {X 0,Y 389.768,Z 589.224,A -85,B 0,C 180,E1 -11597.767,E2 -11597.767} C_VEL
LIN {X 0,Y 389.396,Z 597.196,A -85,B 0,C 180,E1 -11599.601,E2 -11599.601} C_VEL
LIN {X 0,Y 389.329,Z 602.851,A -85,B 0,C 180,E1 -11601.173,E2 -11601.173} C_VEL
LIN {X 0,Y 389.348,Z 608.444,A -85,B 0,C 180,E1 -11603.114,E2 -11603.114} C_VEL
LIN {X 0,Y 389.539,Z 612.226,A -85,B 0,C 180,E1 -11604.823,E2 -11604.823} C_VEL
LIN {X 0,Y 389.579,Z 613.974,A -85,B 0,C 180,E1 -11605.861,E2 -11605.861} C_VEL
LIN {X 0,Y 389.574,Z 616.322,A -85,B 0,C 180,E1 -11607.931,E2 -11607.931} C_VEL
LIN {X 0,Y 389.728,Z 616.957,A -85,B 0,C 180,E1 -11608.966,E2 -11608.966} C_VEL
LIN {X 0,Y 389.828,Z 617.212,A -85,B 0,C 180,E1 -11609.999,E2 -11609.999} C_VEL
LIN {X 0,Y 389.549,Z 616.533,A -85,B 0,C 180,E1 -11612.067,E2 -11612.067} C_VEL
LIN {X 0,Y 389.5,Z 614.393,A -85,B 0,C 180,E1 -11614.138,E2 -11614.138} C_VEL
LIN {X 0,Y 389.398,Z 611.755,A -85,B 0,C 180,E1 -11615.696,E2 -11615.696} C_VEL
LIN {X 0,Y 389.298,Z 608.223,A -85,B 0,C 180,E1 -11617.259,E2 -11617.259} C_VEL
LIN {X 0,Y 389.306,Z 603.661,A -85,B 0,C 180,E1 -11618.826,E2 -11618.826} C_VEL
LIN {X 0,Y 389.509,Z 597.038,A -85,B 0,C 180,E1 -11620.657,E2 -11620.657} C_VEL
LIN {X 0,Y 389.844,Z 588.763,A -85,B 0,C 180,E1 -11622.492,E2 -11622.492} C_VEL
LIN {X 0,Y 390.443,Z 580.12,A -85,B 0,C 180,E1 -11624.062,E2 -11624.062} C_VEL
LIN {X 0,Y 391.277,Z 569.688,A -85,B 0,C 180,E1 -11625.629,E2 -11625.629} C_VEL
LIN {X 0,Y 392.267,Z 559.31,A -85,B 0,C 180,E1 -11626.925,E2 -11626.925} C_VEL
LIN {X 0,Y 393.382,Z 546.751,A -85,B 0,C 180,E1 -11628.218,E2 -11628.218} C_VEL
LIN {X 0,Y 394.393,Z 534.748,A -85,B 0,C 180,E1 -11629.225,E2 -11629.225} C_VEL
LIN {X 0,Y 394.803,Z 526.233,A -85,B 0,C 180,E1 -11629.835,E2 -11629.835} C_VEL
LIN {X 0,Y 393.548,Z 512.009,A -85,B 0,C 180,E1 -11630.719,E2 -11630.719} C_VEL
LIN {X 0,Y 391.767,Z 496.867,A -85,B 0,C 180,E1 -11631.455,E2 -11631.455} C_VEL
LIN {X 0,Y 390.061,Z 483.767,A -85,B 0,C 180,E1 -11631.953,E2 -11631.953} C_VEL
LIN {X 0,Y 390.623,Z 473.279,A -85,B 0,C 180,E1 -11635.01,E2 -11635.01} C_VEL
LIN {X 0,Y 391.413,Z 461.043,A -85,B 0,C 180,E1 -11638.627,E2 -11638.627} C_VEL
LIN {X 0,Y 392.254,Z 450.165,A -85,B 0,C 180,E1 -11641.906,E2 -11641.906} C_VEL
LIN {X 0,Y 393.122,Z 440.418,A -85,B 0,C 180,E1 -11644.893,E2 -11644.893} C_VEL
LIN {X 0,Y 394.293,Z 428.637,A -85,B 0,C 180,E1 -11648.596,E2 -11648.596} C_VEL
LIN {X 0,Y 394.63,Z 424.2,A -85,B 0,C 180,E1 -11650.023,E2 -11650.023} C_VEL
LIN {X 0,Y 393.673,Z 417.911,A -85,B 0,C 180,E1 -11652.195,E2 -11652.195} C_VEL
LIN {X 0,Y 391.559,Z 407.774,A -85,B 0,C 180,E1 -11655.883,E2 -11655.883} C_VEL
LIN {X 0,Y 390.076,Z 400.522,A -85,B 0,C 180,E1 -11658.728,E2 -11658.728} C_VEL
LIN {X 0,Y 390.088,Z 400.52,A -85,B 0,C 180,E1 -11660.908,E2 -11660.908} C_VEL
LIN {X 0,Y 390.077,Z 400.52,A -85,B 0,C 180,E1 -11664.792,E2 -11664.792} C_VEL
LIN {X 0,Y 390.018,Z 400.525,A -85,B 0,C 180,E1 -11668.495,E2 -11668.495} C_VEL
LIN {X 0,Y 390.107,Z 400.514,A -85,B 0,C 180,E1 -11672.069,E2 -11672.069} C_VEL
LIN {X 0,Y 390.07,Z 400.521,A -85,B 0,C 180,E1 -11675.519,E2 -11675.519} C_VEL
LIN {X 0,Y 390.045,Z 400.526,A -85,B 0,C 180,E1 -11678.877,E2 -11678.877} C_VEL
LIN {X 0,Y 390.117,Z 400.512,A -85,B 0,C 180,E1 -11682.166,E2 -11682.166} C_VEL
LIN {X 0,Y 390.136,Z 400.513,A -85,B 0,C 180,E1 -11685.393,E2 -11685.393} C_VEL
LIN {X 0,Y 390.149,Z 400.511,A -85,B 0,C 180,E1 -11688.571,E2 -11688.571} C_VEL
LIN {X 0,Y 390.333,Z 400.485,A -85,B 0,C 180,E1 -11691.993,E2 -11691.993} C_VEL
LIN {X 0,Y 390.218,Z 400.504,A -85,B 0,C 180,E1 -11694.834,E2 -11694.834} C_VEL
LIN {X 0,Y 390.41,Z 400.476,A -85,B 0,C 180,E1 -11697.937,E2 -11697.937} C_VEL
LIN {X 0,Y 390.541,Z 400.46,A -85,B 0,C 180,E1 -11700,E2 -11700} C_VEL
LIN {X 0,Y 390.307,Z 400.493,A -85,B 0,C 180,E1 -11703.097,E2 -11703.097} C_VEL
LIN {X 0,Y 390.3,Z 400.489,A -85,B 0,C 180,E1 -11706.651,E2 -11706.651} C_VEL
LIN {X 0,Y 390.2,Z 400.504,A -85,B 0,C 180,E1 -11709.329,E2 -11709.329} C_VEL
LIN {X 0,Y 390.169,Z 400.509,A -85,B 0,C 180,E1 -11712.483,E2 -11712.483} C_VEL
LIN {X 0,Y 390.13,Z 400.511,A -85,B 0,C 180,E1 -11715.678,E2 -11715.678} C_VEL
LIN {X 0,Y 390.096,Z 400.52,A -85,B 0,C 180,E1 -11718.923,E2 -11718.923} C_VEL
LIN {X 0,Y 390.031,Z 400.525,A -85,B 0,C 180,E1 -11722.235,E2 -11722.235} C_VEL
LIN {X 0,Y 390.11,Z 400.513,A -85,B 0,C 180,E1 -11725.744,E2 -11725.744} C_VEL
LIN {X 0,Y 390.05,Z 400.523,A -85,B 0,C 180,E1 -11729.111,E2 -11729.111} C_VEL
LIN {X 0,Y 390.035,Z 400.528,A -85,B 0,C 180,E1 -11732.723,E2 -11732.723} C_VEL
LIN {X 0,Y 390.05,Z 400.521,A -85,B 0,C 180,E1 -11735.827,E2 -11735.827} C_VEL
LIN {X 0,Y 390.066,Z 400.52,A -85,B 0,C 180,E1 -11739.22,E2 -11739.22} C_VEL
LIN {X 0,Y 390.039,Z 400.526,A -85,B 0,C 180,E1 -11742.376,E2 -11742.376} C_VEL
LIN {X 0,Y 390.041,Z 400.522,A -85,B 0,C 180,E1 -11745.356,E2 -11745.356} C_VEL
LIN {X 0,Y 390.064,Z 400.523,A -85,B 0,C 180,E1 -11748.193,E2 -11748.193} C_VEL
LIN {X 0,Y 390.092,Z 400.518,A -85,B 0,C 180,E1 -11750.91,E2 -11750.91} C_VEL
LIN {X 0,Y 390.083,Z 400.52,A -85,B 0,C 180,E1 -11754.795,E2 -11754.795} C_VEL
LIN {X 0,Y 390.03,Z 400.525,A -85,B 0,C 180,E1 -11757.877,E2 -11757.877} C_VEL
LIN {X 0,Y 390.057,Z 400.522,A -85,B 0,C 180,E1 -11760.892,E2 -11760.892} C_VEL
LIN {X 0,Y 390.119,Z 400.517,A -85,B 0,C 180,E1 -11764.258,E2 -11764.258} C_VEL
LIN {X 0,Y 390.04,Z 400.523,A -85,B 0,C 180,E1 -11767.767,E2 -11767.767} C_VEL
LIN {X 0,Y 390.106,Z 400.514,A -85,B 0,C 180,E1 -11771.079,E2 -11771.079} C_VEL
LIN {X 0,Y 390.122,Z 400.512,A -85,B 0,C 180,E1 -11773.249,E2 -11773.249} C_VEL
LIN {X 0,Y 390.052,Z 400.641,A -85,B 0,C 180,E1 -11774.822,E2 -11774.822} C_VEL
LIN {X 0,Y 394.387,Z 413.649,A -85,B 0,C 180,E1 -11775.459,E2 -11775.459} C_VEL
LIN {X 0,Y 395.862,Z 419.406,A -85,B 0,C 180,E1 -11775.794,E2 -11775.794} C_VEL
LIN {X 0,Y 395.424,Z 431.283,A -85,B 0,C 180,E1 -11776.472,E2 -11776.472} C_VEL
LIN {X 0,Y 394.863,Z 443.523,A -85,B 0,C 180,E1 -11777.408,E2 -11777.408} C_VEL
LIN {X 0,Y 394.177,Z 454.059,A -85,B 0,C 180,E1 -11778.43,E2 -11778.43} C_VEL
LIN {X 0,Y 393.359,Z 464.518,A -85,B 0,C 180,E1 -11779.709,E2 -11779.709} C_VEL
LIN {X 0,Y 392.604,Z 473.019,A -85,B 0,C 180,E1 -11780.99,E2 -11780.99} C_VEL
LIN {X 0,Y 391.958,Z 481.293,A -85,B 0,C 180,E1 -11782.532,E2 -11782.532} C_VEL
LIN {X 0,Y 391.335,Z 486.933,A -85,B 0,C 180,E1 -11783.815,E2 -11783.815} C_VEL
LIN {X 0,Y 390.971,Z 492.411,A -85,B 0,C 180,E1 -11785.361,E2 -11785.361} C_VEL
LIN {X 0,Y 390.573,Z 496.724,A -85,B 0,C 180,E1 -11786.907,E2 -11786.907} C_VEL
LIN {X 0,Y 390.353,Z 498.993,A -85,B 0,C 180,E1 -11787.938,E2 -11787.938} C_VEL
LIN {X 0,Y 390.182,Z 500.851,A -85,B 0,C 180,E1 -11788.969,E2 -11788.969} C_VEL
LIN {X 0,Y 390.084,Z 502.299,A -85,B 0,C 180,E1 -11790.001,E2 -11790.001} C_VEL
LIN {X 0,Y 389.976,Z 503.949,A -85,B 0,C 180,E1 -11792.067,E2 -11792.067} C_VEL
LIN {X 0,Y 389.839,Z 504.237,A -85,B 0,C 180,E1 -11793.101,E2 -11793.101} C_VEL
LIN {X 0,Y 389.916,Z 504.106,A -85,B 0,C 180,E1 -11794.136,E2 -11794.136} C_VEL
LIN {X 0,Y 390.311,Z 502.627,A -85,B 0,C 180,E1 -11796.203,E2 -11796.203} C_VEL
LIN {X 0,Y 390.399,Z 501.344,A -85,B 0,C 180,E1 -11797.24,E2 -11797.24} C_VEL
LIN {X 0,Y 390.709,Z 498.586,A -85,B 0,C 180,E1 -11798.796,E2 -11798.796} C_VEL
LIN {X 0,Y 391.195,Z 494.807,A -85,B 0,C 180,E1 -11800.351,E2 -11800.351} C_VEL
LIN {X 0,Y 391.74,Z 489.907,A -85,B 0,C 180,E1 -11801.908,E2 -11801.908} C_VEL
LIN {X 0,Y 392.323,Z 483.7,A -85,B 0,C 180,E1 -11803.468,E2 -11803.468} C_VEL
LIN {X 0,Y 392.929,Z 477.207,A -85,B 0,C 180,E1 -11804.797,E2 -11804.797} C_VEL
LIN {X 0,Y 393.855,Z 467.96,A -85,B 0,C 180,E1 -11806.324,E2 -11806.324} C_VEL
LIN {X 0,Y 394.683,Z 458.179,A -85,B 0,C 180,E1 -11807.622,E2 -11807.622} C_VEL
LIN {X 0,Y 395.461,Z 447.119,A -85,B 0,C 180,E1 -11808.792,E2 -11808.792} C_VEL
LIN {X 0,Y 395.713,Z 442.921,A -85,B 0,C 180,E1 -11809.169,E2 -11809.169} C_VEL
LIN {X 0,Y 395.465,Z 437.862,A -85,B 0,C 180,E1 -11809.613,E2 -11809.613} C_VEL
LIN {X 0,Y 394.329,Z 432.888,A -85,B 0,C 180,E1 -11810.057,E2 -11810.057} C_VEL
LIN {X 0,Y 390.722,Z 422.973,A -85,B 0,C 180,E1 -11810.893,E2 -11810.893} C_VEL
LIN {X 0,Y 388.328,Z 416.045,A -85,B 0,C 180,E1 -11811.374,E2 -11811.374} C_VEL
LIN {X 0,Y 383.872,Z 404.086,A -85,B 0,C 180,E1 -11812.063,E2 -11812.063} C_VEL
LIN {X 0,Y 382.98,Z 401.404,A -85,B 0,C 180,E1 -11812.198,E2 -11812.198} C_VEL
LIN {X 0,Y 383.057,Z 401.391,A -85,B 0,C 180,E1 -11814.961,E2 -11814.961} C_VEL
LIN {X 0,Y 383.046,Z 401.397,A -85,B 0,C 180,E1 -11818.493,E2 -11818.493} C_VEL
LIN {X 0,Y 383.015,Z 401.402,A -85,B 0,C 180,E1 -11822.15,E2 -11822.15} C_VEL
LIN {X 0,Y 383.023,Z 401.401,A -85,B 0,C 180,E1 -11824.668,E2 -11824.668} C_VEL
LIN {X 0,Y 383.004,Z 401.391,A -85,B 0,C 180,E1 -11827.904,E2 -11827.904} C_VEL
LIN {X 0,Y 382.989,Z 401.401,A -85,B 0,C 180,E1 -11831.348,E2 -11831.348} C_VEL
LIN {X 0,Y 383.003,Z 401.404,A -85,B 0,C 180,E1 -11834.304,E2 -11834.304} C_VEL
LIN {X 0,Y 383.016,Z 401.398,A -85,B 0,C 180,E1 -11837.24,E2 -11837.24} C_VEL
LIN {X 0,Y 383.021,Z 401.376,A -85,B 0,C 180,E1 -11840.414,E2 -11840.414} C_VEL
LIN {X 0,Y 383.032,Z 401.394,A -85,B 0,C 180,E1 -11844.045,E2 -11844.045} C_VEL
LIN {X 0,Y 382.991,Z 401.396,A -85,B 0,C 180,E1 -11847.578,E2 -11847.578} C_VEL
LIN {X 0,Y 382.996,Z 401.368,A -85,B 0,C 180,E1 -11850.3,E2 -11850.3} C_VEL
LIN {X 0,Y 383.085,Z 401.389,A -85,B 0,C 180,E1 -11854.021,E2 -11854.021} C_VEL
LIN {X 0,Y 382.996,Z 401.404,A -85,B 0,C 180,E1 -11857.334,E2 -11857.334} C_VEL
LIN {X 0,Y 383.09,Z 401.529,A -85,B 0,C 180,E1 -11860.246,E2 -11860.246} C_VEL
LIN {X 0,Y 386.895,Z 414.188,A -85,B 0,C 180,E1 -11861.239,E2 -11861.239} C_VEL
LIN {X 0,Y 389.192,Z 422.466,A -85,B 0,C 180,E1 -11861.979,E2 -11861.979} C_VEL
LIN {X 0,Y 388.266,Z 435.813,A -85,B 0,C 180,E1 -11863.165,E2 -11863.165} C_VEL
LIN {X 0,Y 387.316,Z 447.798,A -85,B 0,C 180,E1 -11864.476,E2 -11864.476} C_VEL
LIN {X 0,Y 386.245,Z 459.637,A -85,B 0,C 180,E1 -11866.049,E2 -11866.049} C_VEL
LIN {X 0,Y 385.402,Z 469.426,A -85,B 0,C 180,E1 -11867.627,E2 -11867.627} C_VEL
LIN {X 0,Y 384.794,Z 477.585,A -85,B 0,C 180,E1 -11869.21,E2 -11869.21} C_VEL
LIN {X 0,Y 384.12,Z 485.729,A -85,B 0,C 180,E1 -11871.12,E2 -11871.12} C_VEL
LIN {X 0,Y 383.642,Z 492.583,A -85,B 0,C 180,E1 -11873.161,E2 -11873.161} C_VEL
LIN {X 0,Y 383.228,Z 496.854,A -85,B 0,C 180,E1 -11874.739,E2 -11874.739} C_VEL
LIN {X 0,Y 383.034,Z 499.174,A -85,B 0,C 180,E1 -11875.791,E2 -11875.791} C_VEL
LIN {X 0,Y 382.973,Z 502.687,A -85,B 0,C 180,E1 -11877.896,E2 -11877.896} C_VEL
LIN {X 0,Y 382.997,Z 504.829,A -85,B 0,C 180,E1 -11880,E2 -11880} C_VEL
LIN {X 0,Y 383.161,Z 505.625,A -85,B 0,C 180,E1 -11882.102,E2 -11882.102} C_VEL
LIN {X 0,Y 383.332,Z 505.098,A -85,B 0,C 180,E1 -11884.205,E2 -11884.205} C_VEL
LIN {X 0,Y 383.722,Z 503.238,A -85,B 0,C 180,E1 -11886.309,E2 -11886.309} C_VEL
LIN {X 0,Y 384.403,Z 499.942,A -85,B 0,C 180,E1 -11888.41,E2 -11888.41} C_VEL
LIN {X 0,Y 385.24,Z 495.115,A -85,B 0,C 180,E1 -11890.511,E2 -11890.511} C_VEL
LIN {X 0,Y 386.228,Z 488.663,A -85,B 0,C 180,E1 -11892.612,E2 -11892.612} C_VEL
LIN {X 0,Y 387.404,Z 481.491,A -85,B 0,C 180,E1 -11894.444,E2 -11894.444} C_VEL
LIN {X 0,Y 388.716,Z 473.437,A -85,B 0,C 180,E1 -11896.101,E2 -11896.101} C_VEL
LIN {X 0,Y 390.002,Z 464.809,A -85,B 0,C 180,E1 -11897.568,E2 -11897.568} C_VEL
LIN {X 0,Y 391.277,Z 454.785,A -85,B 0,C 180,E1 -11898.999,E2 -11898.999} C_VEL
LIN {X 0,Y 392.609,Z 443.812,A -85,B 0,C 180,E1 -11900.293,E2 -11900.293} C_VEL
LIN {X 0,Y 393.996,Z 431.15,A -85,B 0,C 180,E1 -11901.516,E2 -11901.516} C_VEL
LIN {X 0,Y 394.11,Z 428.082,A -85,B 0,C 180,E1 -11901.793,E2 -11901.793} C_VEL
LIN {X 0,Y 390.587,Z 417.957,A -85,B 0,C 180,E1 -11903.022,E2 -11903.022} C_VEL
LIN {X 0,Y 385.024,Z 405.523,A -85,B 0,C 180,E1 -11904.525,E2 -11904.525} C_VEL
LIN {X 0,Y 383.362,Z 402.826,A -85,B 0,C 180,E1 -11904.893,E2 -11904.893} C_VEL
LIN {X 0,Y 383.043,Z 401.402,A -85,B 0,C 180,E1 -11905.024,E2 -11905.024} C_VEL
LIN {X 0,Y 383.02,Z 401.398,A -85,B 0,C 180,E1 -11908.494,E2 -11908.494} C_VEL
LIN {X 0,Y 383.012,Z 401.4,A -85,B 0,C 180,E1 -11912.149,E2 -11912.149} C_VEL
LIN {X 0,Y 383.021,Z 401.4,A -85,B 0,C 180,E1 -11914.667,E2 -11914.667} C_VEL
LIN {X 0,Y 383.002,Z 401.402,A -85,B 0,C 180,E1 -11917.903,E2 -11917.903} C_VEL
LIN {X 0,Y 383.033,Z 401.402,A -85,B 0,C 180,E1 -11919.348,E2 -11919.348} C_VEL
LIN {X 0,Y 383.903,Z 405.696,A -85,B 0,C 180,E1 -11922.637,E2 -11922.637} C_VEL
LIN {X 0,Y 384.886,Z 410.213,A -85,B 0,C 180,E1 -11925.409,E2 -11925.409} C_VEL
LIN {X 0,Y 386.003,Z 415.858,A -85,B 0,C 180,E1 -11928.287,E2 -11928.287} C_VEL
LIN {X 0,Y 386.574,Z 419.186,A -85,B 0,C 180,E1 -11929.78,E2 -11929.78} C_VEL
LIN {X 0,Y 386.388,Z 422.426,A -85,B 0,C 180,E1 -11931.064,E2 -11931.064} C_VEL
LIN {X 0,Y 384.807,Z 434.383,A -85,B 0,C 180,E1 -11935.272,E2 -11935.272} C_VEL
LIN {X 0,Y 384.079,Z 444.603,A -85,B 0,C 180,E1 -11938.566,E2 -11938.566} C_VEL
LIN {X 0,Y 383.499,Z 454.599,A -85,B 0,C 180,E1 -11941.6,E2 -11941.6} C_VEL
LIN {X 0,Y 383.023,Z 466.448,A -85,B 0,C 180,E1 -11945.037,E2 -11945.037} C_VEL
LIN {X 0,Y 382.993,Z 467.662,A -85,B 0,C 180,E1 -11945.379,E2 -11945.379} C_VEL
LIN {X 0,Y 383.932,Z 471.998,A -85,B 0,C 180,E1 -11945.645,E2 -11945.645} C_VEL
LIN {X 0,Y 387.027,Z 488.266,A -85,B 0,C 180,E1 -11946.668,E2 -11946.668} C_VEL
LIN {X 0,Y 388.453,Z 502.613,A -85,B 0,C 180,E1 -11947.603,E2 -11947.603} C_VEL
LIN {X 0,Y 388.571,Z 517.869,A -85,B 0,C 180,E1 -11948.682,E2 -11948.682} C_VEL
LIN {X 0,Y 388.494,Z 532.264,A -85,B 0,C 180,E1 -11949.896,E2 -11949.896} C_VEL
LIN {X 0,Y 386.838,Z 545.842,A -85,B 0,C 180,E1 -11951.186,E2 -11951.186} C_VEL
LIN {X 0,Y 385.438,Z 558.314,A -85,B 0,C 180,E1 -11952.627,E2 -11952.627} C_VEL
LIN {X 0,Y 384.29,Z 568.89,A -85,B 0,C 180,E1 -11954.077,E2 -11954.077} C_VEL
LIN {X 0,Y 383.329,Z 580.211,A -85,B 0,C 180,E1 -11955.94,E2 -11955.94} C_VEL
LIN {X 0,Y 382.743,Z 588.333,A -85,B 0,C 180,E1 -11957.539,E2 -11957.539} C_VEL
LIN {X 0,Y 382.359,Z 596.258,A -85,B 0,C 180,E1 -11959.407,E2 -11959.407} C_VEL
LIN {X 0,Y 382.251,Z 601.866,A -85,B 0,C 180,E1 -11961.008,E2 -11961.008} C_VEL
LIN {X 0,Y 382.285,Z 607.697,A -85,B 0,C 180,E1 -11963.094,E2 -11963.094} C_VEL
LIN {X 0,Y 382.462,Z 611.188,A -85,B 0,C 180,E1 -11964.727,E2 -11964.727} C_VEL
LIN {X 0,Y 382.543,Z 612.935,A -85,B 0,C 180,E1 -11965.785,E2 -11965.785} C_VEL
LIN {X 0,Y 382.543,Z 615.261,A -85,B 0,C 180,E1 -11967.893,E2 -11967.893} C_VEL
LIN {X 0,Y 382.71,Z 615.888,A -85,B 0,C 180,E1 -11968.947,E2 -11968.947} C_VEL
LIN {X 0,Y 382.828,Z 616.135,A -85,B 0,C 180,E1 -11969.999,E2 -11969.999} C_VEL
LIN {X 0,Y 382.525,Z 615.426,A -85,B 0,C 180,E1 -11972.105,E2 -11972.105} C_VEL
LIN {X 0,Y 382.467,Z 613.252,A -85,B 0,C 180,E1 -11974.214,E2 -11974.214} C_VEL
